LIN {X 0,Y 573.173,Z 473.905,A -85,B 0,C 180,E1 -2067.979,E2 -2067.979} C_VEL
LIN {X 0,Y 573.326,Z 473.883,A -85,B 0,C 180,E1 -2070,E2 -2070} C_VEL
LIN {X 0,Y 573.306,Z 473.888,A -85,B 0,C 180,E1 -2072.81,E2 -2072.81} C_VEL
LIN {X 0,Y 573.299,Z 473.886,A -85,B 0,C 180,E1 -2075.628,E2 -2075.628} C_VEL
LIN {X 0,Y 573.287,Z 473.888,A -85,B 0,C 180,E1 -2078.459,E2 -2078.459} C_VEL
LIN {X 0,Y 573.274,Z 473.891,A -85,B 0,C 180,E1 -2081.312,E2 -2081.312} C_VEL
LIN {X 0,Y 573.283,Z 473.889,A -85,B 0,C 180,E1 -2084.424,E2 -2084.424} C_VEL
LIN {X 0,Y 573.261,Z 473.893,A -85,B 0,C 180,E1 -2087.111,E2 -2087.111} C_VEL
LIN {X 0,Y 573.255,Z 473.892,A -85,B 0,C 180,E1 -2090.076,E2 -2090.076} C_VEL
LIN {X 0,Y 573.235,Z 473.896,A -85,B 0,C 180,E1 -2093.099,E2 -2093.099} C_VEL
LIN {X 0,Y 573.258,Z 473.894,A -85,B 0,C 180,E1 -2095.409,E2 -2095.409} C_VEL
LIN {X 0,Y 573.253,Z 473.893,A -85,B 0,C 180,E1 -2098.029,E2 -2098.029} C_VEL
LIN {X 0,Y 573.246,Z 473.893,A -85,B 0,C 180,E1 -2100.885,E2 -2100.885} C_VEL
LIN {X 0,Y 573.262,Z 473.893,A -85,B 0,C 180,E1 -2103.524,E2 -2103.524} C_VEL
LIN {X 0,Y 573.261,Z 473.894,A -85,B 0,C 180,E1 -2106.048,E2 -2106.048} C_VEL
LIN {X 0,Y 573.249,Z 473.892,A -85,B 0,C 180,E1 -2108.7,E2 -2108.7} C_VEL
LIN {X 0,Y 573.228,Z 473.895,A -85,B 0,C 180,E1 -2111.457,E2 -2111.457} C_VEL
LIN {X 0,Y 573.238,Z 473.896,A -85,B 0,C 180,E1 -2114.333,E2 -2114.333} C_VEL
LIN {X 0,Y 573.243,Z 473.893,A -85,B 0,C 180,E1 -2117.358,E2 -2117.358} C_VEL
LIN {X 0,Y 573.273,Z 473.889,A -85,B 0,C 180,E1 -2119.477,E2 -2119.477} C_VEL
LIN {X 0,Y 573.235,Z 473.895,A -85,B 0,C 180,E1 -2122.192,E2 -2122.192} C_VEL
LIN {X 0,Y 573.236,Z 473.894,A -85,B 0,C 180,E1 -2125.228,E2 -2125.228} C_VEL
LIN {X 0,Y 573.256,Z 473.891,A -85,B 0,C 180,E1 -2127.77,E2 -2127.77} C_VEL
LIN {X 0,Y 573.263,Z 473.893,A -85,B 0,C 180,E1 -2130.634,E2 -2130.634} C_VEL
LIN {X 0,Y 573.27,Z 473.89,A -85,B 0,C 180,E1 -2133.5,E2 -2133.5} C_VEL
LIN {X 0,Y 573.23,Z 473.895,A -85,B 0,C 180,E1 -2136.134,E2 -2136.134} C_VEL
LIN {X 0,Y 573.26,Z 473.893,A -85,B 0,C 180,E1 -2139.174,E2 -2139.174} C_VEL
LIN {X 0,Y 573.229,Z 473.898,A -85,B 0,C 180,E1 -2141.411,E2 -2141.411} C_VEL
LIN {X 0,Y 573.253,Z 473.893,A -85,B 0,C 180,E1 -2143.622,E2 -2143.622} C_VEL
LIN {X 0,Y 573.272,Z 473.89,A -85,B 0,C 180,E1 -2145.807,E2 -2145.807} C_VEL
LIN {X 0,Y 573.261,Z 473.892,A -85,B 0,C 180,E1 -2148.745,E2 -2148.745} C_VEL
LIN {X 0,Y 573.29,Z 473.887,A -85,B 0,C 180,E1 -2151.541,E2 -2151.541} C_VEL
LIN {X 0,Y 573.289,Z 473.891,A -85,B 0,C 180,E1 -2154.372,E2 -2154.372} C_VEL
LIN {X 0,Y 573.312,Z 473.887,A -85,B 0,C 180,E1 -2157.892,E2 -2157.892} C_VEL
LIN {X 0,Y 573.332,Z 473.882,A -85,B 0,C 180,E1 -2160.702,E2 -2160.702} C_VEL
LIN {X 0,Y 573.24,Z 473.894,A -85,B 0,C 180,E1 -2163.514,E2 -2163.514} C_VEL
LIN {X 0,Y 573.294,Z 473.887,A -85,B 0,C 180,E1 -2165.628,E2 -2165.628} C_VEL
LIN {X 0,Y 573.288,Z 473.89,A -85,B 0,C 180,E1 -2168.459,E2 -2168.459} C_VEL
LIN {X 0,Y 573.27,Z 473.89,A -85,B 0,C 180,E1 -2171.312,E2 -2171.312} C_VEL
LIN {X 0,Y 573.271,Z 473.89,A -85,B 0,C 180,E1 -2174.193,E2 -2174.193} C_VEL
LIN {X 0,Y 573.259,Z 473.892,A -85,B 0,C 180,E1 -2177.112,E2 -2177.112} C_VEL
LIN {X 0,Y 573.251,Z 473.893,A -85,B 0,C 180,E1 -2180.077,E2 -2180.077} C_VEL
LIN {X 0,Y 573.232,Z 473.895,A -85,B 0,C 180,E1 -2183.099,E2 -2183.099} C_VEL
LIN {X 0,Y 573.253,Z 473.893,A -85,B 0,C 180,E1 -2185.41,E2 -2185.41} C_VEL
LIN {X 0,Y 573.251,Z 473.892,A -85,B 0,C 180,E1 -2188.03,E2 -2188.03} C_VEL
LIN {X 0,Y 573.255,Z 473.892,A -85,B 0,C 180,E1 -2190.176,E2 -2190.176} C_VEL
LIN {X 0,Y 573.255,Z 473.891,A -85,B 0,C 180,E1 -2192.645,E2 -2192.645} C_VEL
LIN {X 0,Y 573.267,Z 473.89,A -85,B 0,C 180,E1 -2195.184,E2 -2195.184} C_VEL
LIN {X 0,Y 573.236,Z 473.895,A -85,B 0,C 180,E1 -2197.807,E2 -2197.807} C_VEL
LIN {X 0,Y 573.268,Z 473.893,A -85,B 0,C 180,E1 -2200.528,E2 -2200.528} C_VEL
LIN {X 0,Y 573.254,Z 473.892,A -85,B 0,C 180,E1 -2203.671,E2 -2203.671} C_VEL
LIN {X 0,Y 573.238,Z 473.895,A -85,B 0,C 180,E1 -2206.641,E2 -2206.641} C_VEL
LIN {X 0,Y 573.272,Z 473.89,A -85,B 0,C 180,E1 -2209.478,E2 -2209.478} C_VEL
LIN {X 0,Y 573.235,Z 473.896,A -85,B 0,C 180,E1 -2212.193,E2 -2212.193} C_VEL
LIN {X 0,Y 573.269,Z 473.892,A -85,B 0,C 180,E1 -2214.817,E2 -2214.817} C_VEL
LIN {X 0,Y 573.253,Z 473.894,A -85,B 0,C 180,E1 -2217.355,E2 -2217.355} C_VEL
LIN {X 0,Y 573.27,Z 473.92,A -85,B 0,C 180,E1 -2218.113,E2 -2218.113} C_VEL
LIN {X 0,Y 573.657,Z 478.198,A -85,B 0,C 180,E1 -2219.447,E2 -2219.447} C_VEL
LIN {X 0,Y 573.521,Z 487.647,A -85,B 0,C 180,E1 -2222.248,E2 -2222.248} C_VEL
LIN {X 0,Y 573.466,Z 497.583,A -85,B 0,C 180,E1 -2225.079,E2 -2225.079} C_VEL
LIN {X 0,Y 573.37,Z 508.135,A -85,B 0,C 180,E1 -2228.047,E2 -2228.047} C_VEL
LIN {X 0,Y 573.251,Z 519.115,A -85,B 0,C 180,E1 -2231.072,E2 -2231.072} C_VEL
LIN {X 0,Y 573.175,Z 529.877,A -85,B 0,C 180,E1 -2233.986,E2 -2233.986} C_VEL
LIN {X 0,Y 573.105,Z 540.748,A -85,B 0,C 180,E1 -2236.888,E2 -2236.888} C_VEL
LIN {X 0,Y 573.057,Z 550.26,A -85,B 0,C 180,E1 -2239.4,E2 -2239.4} C_VEL
LIN {X 0,Y 573.08,Z 553.109,A -85,B 0,C 180,E1 -2240.125,E2 -2240.125} C_VEL
LIN {X 0,Y 573.479,Z 559.596,A -85,B 0,C 180,E1 -2240.277,E2 -2240.277} C_VEL
LIN {X 0,Y 573.449,Z 568.903,A -85,B 0,C 180,E1 -2240.566,E2 -2240.566} C_VEL
LIN {X 0,Y 573.402,Z 577.409,A -85,B 0,C 180,E1 -2240.921,E2 -2240.921} C_VEL
LIN {X 0,Y 573.339,Z 585.736,A -85,B 0,C 180,E1 -2241.364,E2 -2241.364} C_VEL
LIN {X 0,Y 573.252,Z 593.772,A -85,B 0,C 180,E1 -2241.895,E2 -2241.895} C_VEL
LIN {X 0,Y 573.187,Z 601.421,A -85,B 0,C 180,E1 -2242.515,E2 -2242.515} C_VEL
LIN {X 0,Y 573.155,Z 609.552,A -85,B 0,C 180,E1 -2243.323,E2 -2243.323} C_VEL
LIN {X 0,Y 573.112,Z 616.435,A -85,B 0,C 180,E1 -2244.194,E2 -2244.194} C_VEL
LIN {X 0,Y 573.005,Z 621.989,A -85,B 0,C 180,E1 -2245.075,E2 -2245.075} C_VEL
LIN {X 0,Y 573.036,Z 627.149,A -85,B 0,C 180,E1 -2246.133,E2 -2246.133} C_VEL
LIN {X 0,Y 572.992,Z 629.79,A -85,B 0,C 180,E1 -2246.836,E2 -2246.836} C_VEL
LIN {X 0,Y 572.939,Z 632.682,A -85,B 0,C 180,E1 -2247.891,E2 -2247.891} C_VEL
LIN {X 0,Y 572.945,Z 633.937,A -85,B 0,C 180,E1 -2248.595,E2 -2248.595} C_VEL
LIN {X 0,Y 572.938,Z 634.711,A -85,B 0,C 180,E1 -2249.298,E2 -2249.298} C_VEL
LIN {X 0,Y 572.935,Z 635,A -85,B 0,C 180,E1 -2250,E2 -2250} C_VEL
LIN {X 0,Y 572.938,Z 634.711,A -85,B 0,C 180,E1 -2250.703,E2 -2250.703} C_VEL
LIN {X 0,Y 572.945,Z 633.936,A -85,B 0,C 180,E1 -2251.406,E2 -2251.406} C_VEL
LIN {X 0,Y 572.939,Z 632.68,A -85,B 0,C 180,E1 -2252.109,E2 -2252.109} C_VEL
LIN {X 0,Y 572.992,Z 629.787,A -85,B 0,C 180,E1 -2253.164,E2 -2253.164} C_VEL
LIN {X 0,Y 573.024,Z 627.146,A -85,B 0,C 180,E1 -2253.868,E2 -2253.868} C_VEL
LIN {X 0,Y 573.005,Z 621.984,A -85,B 0,C 180,E1 -2254.926,E2 -2254.926} C_VEL
LIN {X 0,Y 573.137,Z 615.184,A -85,B 0,C 180,E1 -2255.983,E2 -2255.983} C_VEL
LIN {X 0,Y 573.164,Z 607.801,A -85,B 0,C 180,E1 -2256.86,E2 -2256.86} C_VEL
LIN {X 0,Y 573.213,Z 600.402,A -85,B 0,C 180,E1 -2257.574,E2 -2257.574} C_VEL
LIN {X 0,Y 573.275,Z 592.542,A -85,B 0,C 180,E1 -2258.194,E2 -2258.194} C_VEL
LIN {X 0,Y 573.385,Z 582.727,A -85,B 0,C 180,E1 -2258.814,E2 -2258.814} C_VEL
LIN {X 0,Y 573.429,Z 571.291,A -85,B 0,C 180,E1 -2259.346,E2 -2259.346} C_VEL
LIN {X 0,Y 573.507,Z 561.233,A -85,B 0,C 180,E1 -2259.679,E2 -2259.679} C_VEL
LIN {X 0,Y 573.212,Z 555.017,A -85,B 0,C 180,E1 -2259.84,E2 -2259.84} C_VEL
LIN {X 0,Y 573.019,Z 553.301,A -85,B 0,C 180,E1 -2259.887,E2 -2259.887} C_VEL
LIN {X 0,Y 573.067,Z 544.36,A -85,B 0,C 180,E1 -2262.393,E2 -2262.393} C_VEL
LIN {X 0,Y 573.155,Z 534.141,A -85,B 0,C 180,E1 -2265.286,E2 -2265.286} C_VEL
LIN {X 0,Y 573.21,Z 523.922,A -85,B 0,C 180,E1 -2268.219,E2 -2268.219} C_VEL
LIN {X 0,Y 573.273,Z 514.981,A -85,B 0,C 180,E1 -2270.826,E2 -2270.826} C_VEL
LIN {X 0,Y 573.346,Z 506.041,A -85,B 0,C 180,E1 -2273.477,E2 -2273.477} C_VEL
LIN {X 0,Y 573.412,Z 496.934,A -85,B 0,C 180,E1 -2276.183,E2 -2276.183} C_VEL
LIN {X 0,Y 573.474,Z 487.899,A -85,B 0,C 180,E1 -2278.952,E2 -2278.952} C_VEL
LIN {X 0,Y 573.623,Z 480.281,A -85,B 0,C 180,E1 -2281.38,E2 -2281.38} C_VEL
LIN {X 0,Y 573.54,Z 475.462,A -85,B 0,C 180,E1 -2283.045,E2 -2283.045} C_VEL
LIN {X 0,Y 573.29,Z 473.89,A -85,B 0,C 180,E1 -2283.692,E2 -2283.692} C_VEL
LIN {X 0,Y 573.24,Z 473.893,A -85,B 0,C 180,E1 -2286.05,E2 -2286.05} C_VEL
LIN {X 0,Y 573.25,Z 473.896,A -85,B 0,C 180,E1 -2288.701,E2 -2288.701} C_VEL
LIN {X 0,Y 573.232,Z 473.894,A -85,B 0,C 180,E1 -2291.457,E2 -2291.457} C_VEL
LIN {X 0,Y 573.238,Z 473.891,A -85,B 0,C 180,E1 -2294.334,E2 -2294.334} C_VEL
LIN {X 0,Y 573.246,Z 473.89,A -85,B 0,C 180,E1 -2297.358,E2 -2297.358} C_VEL
LIN {X 0,Y 573.243,Z 473.891,A -85,B 0,C 180,E1 -2300.393,E2 -2300.393} C_VEL
LIN {X 0,Y 573.255,Z 473.894,A -85,B 0,C 180,E1 -2303.078,E2 -2303.078} C_VEL
LIN {X 0,Y 573.269,Z 473.889,A -85,B 0,C 180,E1 -2305.672,E2 -2305.672} C_VEL
LIN {X 0,Y 573.141,Z 473.909,A -85,B 0,C 180,E1 -2308.178,E2 -2308.178} C_VEL
LIN {X 0,Y 573.099,Z 477.229,A -85,B 0,C 180,E1 -2310.625,E2 -2310.625} C_VEL
LIN {X 0,Y 573.045,Z 480.484,A -85,B 0,C 180,E1 -2313.014,E2 -2313.014} C_VEL
LIN {X 0,Y 573.025,Z 483.626,A -85,B 0,C 180,E1 -2315.355,E2 -2315.355} C_VEL
LIN {X 0,Y 572.985,Z 486.997,A -85,B 0,C 180,E1 -2317.652,E2 -2317.652} C_VEL
LIN {X 0,Y 573.021,Z 491.592,A -85,B 0,C 180,E1 -2320.661,E2 -2320.661} C_VEL
LIN {X 0,Y 572.976,Z 496.187,A -85,B 0,C 180,E1 -2323.614,E2 -2323.614} C_VEL
LIN {X 0,Y 572.993,Z 500.783,A -85,B 0,C 180,E1 -2326.524,E2 -2326.524} C_VEL
LIN {X 0,Y 572.98,Z 505.378,A -85,B 0,C 180,E1 -2329.398,E2 -2329.398} C_VEL
LIN {X 0,Y 572.976,Z 506.707,A -85,B 0,C 180,E1 -2330.224,E2 -2330.224} C_VEL
LIN {X 0,Y 573.49,Z 512.89,A -85,B 0,C 180,E1 -2330.411,E2 -2330.411} C_VEL
LIN {X 0,Y 573.429,Z 524.583,A -85,B 0,C 180,E1 -2330.832,E2 -2330.832} C_VEL
LIN {X 0,Y 573.333,Z 534.974,A -85,B 0,C 180,E1 -2331.364,E2 -2331.364} C_VEL
LIN {X 0,Y 573.246,Z 543.153,A -85,B 0,C 180,E1 -2331.895,E2 -2331.895} C_VEL
LIN {X 0,Y 573.196,Z 550.906,A -85,B 0,C 180,E1 -2332.515,E2 -2332.515} C_VEL
LIN {X 0,Y 573.167,Z 557.376,A -85,B 0,C 180,E1 -2333.141,E2 -2333.141} C_VEL
LIN {X 0,Y 573.138,Z 564.834,A -85,B 0,C 180,E1 -2334.017,E2 -2334.017} C_VEL
LIN {X 0,Y 573.004,Z 571.741,A -85,B 0,C 180,E1 -2335.075,E2 -2335.075} C_VEL
LIN {X 0,Y 573.033,Z 575.438,A -85,B 0,C 180,E1 -2335.78,E2 -2335.78} C_VEL
LIN {X 0,Y 573.053,Z 578.452,A -85,B 0,C 180,E1 -2336.484,E2 -2336.484} C_VEL
LIN {X 0,Y 572.962,Z 580.787,A -85,B 0,C 180,E1 -2337.188,E2 -2337.188} C_VEL
LIN {X 0,Y 572.937,Z 582.578,A -85,B 0,C 180,E1 -2337.891,E2 -2337.891} C_VEL
LIN {X 0,Y 572.946,Z 583.874,A -85,B 0,C 180,E1 -2338.594,E2 -2338.594} C_VEL
LIN {X 0,Y 572.937,Z 584.69,A -85,B 0,C 180,E1 -2339.297,E2 -2339.297} C_VEL
LIN {X 0,Y 572.934,Z 584.996,A -85,B 0,C 180,E1 -2340,E2 -2340} C_VEL
LIN {X 0,Y 572.939,Z 584.731,A -85,B 0,C 180,E1 -2340.703,E2 -2340.703} C_VEL
LIN {X 0,Y 572.945,Z 583.997,A -85,B 0,C 180,E1 -2341.406,E2 -2341.406} C_VEL
LIN {X 0,Y 572.939,Z 582.783,A -85,B 0,C 180,E1 -2342.109,E2 -2342.109} C_VEL
LIN {X 0,Y 572.98,Z 579.935,A -85,B 0,C 180,E1 -2343.164,E2 -2343.164} C_VEL
LIN {X 0,Y 573.026,Z 577.341,A -85,B 0,C 180,E1 -2343.868,E2 -2343.868} C_VEL
LIN {X 0,Y 572.984,Z 572.231,A -85,B 0,C 180,E1 -2344.925,E2 -2344.925} C_VEL
LIN {X 0,Y 573.113,Z 566.733,A -85,B 0,C 180,E1 -2345.807,E2 -2345.807} C_VEL
LIN {X 0,Y 573.157,Z 558.342,A -85,B 0,C 180,E1 -2346.849,E2 -2346.849} C_VEL
LIN {X 0,Y 573.213,Z 550.917,A -85,B 0,C 180,E1 -2347.574,E2 -2347.574} C_VEL
LIN {X 0,Y 573.274,Z 543.167,A -85,B 0,C 180,E1 -2348.194,E2 -2348.194} C_VEL
LIN {X 0,Y 573.386,Z 534.991,A -85,B 0,C 180,E1 -2348.724,E2 -2348.724} C_VEL
LIN {X 0,Y 573.394,Z 526.474,A -85,B 0,C 180,E1 -2349.169,E2 -2349.169} C_VEL
LIN {X 0,Y 573.488,Z 515.241,A -85,B 0,C 180,E1 -2349.612,E2 -2349.612} C_VEL
LIN {X 0,Y 573.182,Z 508.35,A -85,B 0,C 180,E1 -2349.806,E2 -2349.806} C_VEL
LIN {X 0,Y 572.968,Z 506.482,A -85,B 0,C 180,E1 -2349.888,E2 -2349.888} C_VEL
LIN {X 0,Y 572.967,Z 501.591,A -85,B 0,C 180,E1 -2352.755,E2 -2352.755} C_VEL
LIN {X 0,Y 572.988,Z 497.923,A -85,B 0,C 180,E1 -2354.926,E2 -2354.926} C_VEL
LIN {X 0,Y 572.967,Z 493.032,A -85,B 0,C 180,E1 -2357.857,E2 -2357.857} C_VEL
LIN {X 0,Y 572.998,Z 489.364,A -85,B 0,C 180,E1 -2360.086,E2 -2360.086} C_VEL
LIN {X 0,Y 573,Z 488.115,A -85,B 0,C 180,E1 -2360.852,E2 -2360.852} C_VEL
LIN {X 0,Y 572.335,Z 487.218,A -85,B 0,C 180,E1 -2361.432,E2 -2361.432} C_VEL
LIN {X 0,Y 569.468,Z 485.896,A -85,B 0,C 180,E1 -2362.375,E2 -2362.375} C_VEL
LIN {X 0,Y 567.048,Z 484.865,A -85,B 0,C 180,E1 -2363.135,E2 -2363.135} C_VEL
LIN {X 0,Y 566.015,Z 484.027,A -85,B 0,C 180,E1 -2363.72,E2 -2363.72} C_VEL
LIN {X 0,Y 565.934,Z 483.727,A -85,B 0,C 180,E1 -2363.918,E2 -2363.918} C_VEL
LIN {X 0,Y 566.026,Z 479.241,A -85,B 0,C 180,E1 -2366.912,E2 -2366.912} C_VEL
LIN {X 0,Y 566.051,Z 478.708,A -85,B 0,C 180,E1 -2367.293,E2 -2367.293} C_VEL
LIN {X 0,Y 566.076,Z 484.914,A -85,B 0,C 180,E1 -2369.776,E2 -2369.776} C_VEL
LIN {X 0,Y 566.114,Z 491.47,A -85,B 0,C 180,E1 -2372.415,E2 -2372.415} C_VEL
LIN {X 0,Y 566.048,Z 497.672,A -85,B 0,C 180,E1 -2374.97,E2 -2374.97} C_VEL
LIN {X 0,Y 566.002,Z 504.801,A -85,B 0,C 180,E1 -2377.926,E2 -2377.926} C_VEL
LIN {X 0,Y 565.959,Z 511.741,A -85,B 0,C 180,E1 -2380.756,E2 -2380.756} C_VEL
LIN {X 0,Y 565.94,Z 518.557,A -85,B 0,C 180,E1 -2383.5,E2 -2383.5} C_VEL
LIN {X 0,Y 565.921,Z 525.026,A -85,B 0,C 180,E1 -2386.078,E2 -2386.078} C_VEL
LIN {X 0,Y 566.504,Z 532.234,A -85,B 0,C 180,E1 -2386.273,E2 -2386.273} C_VEL
LIN {X 0,Y 566.445,Z 541.756,A -85,B 0,C 180,E1 -2386.602,E2 -2386.602} C_VEL
LIN {X 0,Y 566.326,Z 552.862,A -85,B 0,C 180,E1 -2387.126,E2 -2387.126} C_VEL
LIN {X 0,Y 566.235,Z 563.213,A -85,B 0,C 180,E1 -2387.794,E2 -2387.794} C_VEL
LIN {X 0,Y 566.159,Z 571.873,A -85,B 0,C 180,E1 -2388.504,E2 -2388.504} C_VEL
LIN {X 0,Y 566.031,Z 580.29,A -85,B 0,C 180,E1 -2389.375,E2 -2389.375} C_VEL
LIN {X 0,Y 565.996,Z 587.634,A -85,B 0,C 180,E1 -2390.341,E2 -2390.341} C_VEL
LIN {X 0,Y 565.922,Z 594.266,A -85,B 0,C 180,E1 -2391.479,E2 -2391.479} C_VEL
LIN {X 0,Y 565.906,Z 599.119,A -85,B 0,C 180,E1 -2392.638,E2 -2392.638} C_VEL
LIN {X 0,Y 565.859,Z 602.529,A -85,B 0,C 180,E1 -2393.833,E2 -2393.833} C_VEL
LIN {X 0,Y 565.849,Z 604.519,A -85,B 0,C 180,E1 -2395.059,E2 -2395.059} C_VEL
LIN {X 0,Y 565.85,Z 604.904,A -85,B 0,C 180,E1 -2396.321,E2 -2396.321} C_VEL
LIN {X 0,Y 565.826,Z 604.648,A -85,B 0,C 180,E1 -2396.871,E2 -2396.871} C_VEL
LIN {X 0,Y 565.853,Z 603.582,A -85,B 0,C 180,E1 -2397.719,E2 -2397.719} C_VEL
LIN {X 0,Y 565.898,Z 600.701,A -85,B 0,C 180,E1 -2398.973,E2 -2398.973} C_VEL
LIN {X 0,Y 565.908,Z 597.854,A -85,B 0,C 180,E1 -2399.803,E2 -2399.803} C_VEL
LIN {X 0,Y 565.95,Z 593.777,A -85,B 0,C 180,E1 -2400.705,E2 -2400.705} C_VEL
LIN {X 0,Y 565.974,Z 588.203,A -85,B 0,C 180,E1 -2401.663,E2 -2401.663} C_VEL
LIN {X 0,Y 566.056,Z 582.479,A -85,B 0,C 180,E1 -2402.452,E2 -2402.452} C_VEL
LIN {X 0,Y 566.094,Z 574.222,A -85,B 0,C 180,E1 -2403.364,E2 -2403.364} C_VEL
LIN {X 0,Y 566.169,Z 566.419,A -85,B 0,C 180,E1 -2404.051,E2 -2404.051} C_VEL
LIN {X 0,Y 566.267,Z 558.201,A -85,B 0,C 180,E1 -2404.638,E2 -2404.638} C_VEL
LIN {X 0,Y 566.343,Z 549.386,A -85,B 0,C 180,E1 -2405.142,E2 -2405.142} C_VEL
LIN {X 0,Y 566.465,Z 540.46,A -85,B 0,C 180,E1 -2405.539,E2 -2405.539} C_VEL
LIN {X 0,Y 566.5,Z 530.802,A -85,B 0,C 180,E1 -2405.857,E2 -2405.857} C_VEL
LIN {X 0,Y 565.895,Z 525.251,A -85,B 0,C 180,E1 -2406.024,E2 -2406.024} C_VEL
LIN {X 0,Y 565.906,Z 518.495,A -85,B 0,C 180,E1 -2408.89,E2 -2408.89} C_VEL
LIN {X 0,Y 565.962,Z 513.187,A -85,B 0,C 180,E1 -2411.164,E2 -2411.164} C_VEL
LIN {X 0,Y 565.98,Z 506.312,A -85,B 0,C 180,E1 -2414.146,E2 -2414.146} C_VEL
LIN {X 0,Y 566.01,Z 501.294,A -85,B 0,C 180,E1 -2416.354,E2 -2416.354} C_VEL
LIN {X 0,Y 566.056,Z 494.758,A -85,B 0,C 180,E1 -2419.266,E2 -2419.266} C_VEL
LIN {X 0,Y 566.065,Z 488.079,A -85,B 0,C 180,E1 -2422.15,E2 -2422.15} C_VEL
LIN {X 0,Y 566.126,Z 481.423,A -85,B 0,C 180,E1 -2425.014,E2 -2425.014} C_VEL
LIN {X 0,Y 566.113,Z 474.784,A -85,B 0,C 180,E1 -2427.954,E2 -2427.954} C_VEL
LIN {X 0,Y 566.296,Z 474.758,A -85,B 0,C 180,E1 -2430,E2 -2430} C_VEL
LIN {X 0,Y 566.272,Z 474.764,A -85,B 0,C 180,E1 -2432.845,E2 -2432.845} C_VEL
LIN {X 0,Y 566.267,Z 474.762,A -85,B 0,C 180,E1 -2435.698,E2 -2435.698} C_VEL
LIN {X 0,Y 566.23,Z 474.768,A -85,B 0,C 180,E1 -2438.565,E2 -2438.565} C_VEL
LIN {X 0,Y 566.244,Z 474.766,A -85,B 0,C 180,E1 -2441.454,E2 -2441.454} C_VEL
LIN {X 0,Y 566.236,Z 474.767,A -85,B 0,C 180,E1 -2444.506,E2 -2444.506} C_VEL
LIN {X 0,Y 566.205,Z 474.771,A -85,B 0,C 180,E1 -2447.331,E2 -2447.331} C_VEL
LIN {X 0,Y 566.216,Z 474.769,A -85,B 0,C 180,E1 -2450.337,E2 -2450.337} C_VEL
LIN {X 0,Y 566.191,Z 474.771,A -85,B 0,C 180,E1 -2453.403,E2 -2453.403} C_VEL
LIN {X 0,Y 566.226,Z 474.767,A -85,B 0,C 180,E1 -2455.748,E2 -2455.748} C_VEL
LIN {X 0,Y 566.202,Z 474.77,A -85,B 0,C 180,E1 -2458.202,E2 -2458.202} C_VEL
LIN {X 0,Y 566.196,Z 474.771,A -85,B 0,C 180,E1 -2460.591,E2 -2460.591} C_VEL
LIN {X 0,Y 566.23,Z 474.766,A -85,B 0,C 180,E1 -2463.101,E2 -2463.101} C_VEL
LIN {X 0,Y 566.213,Z 474.769,A -85,B 0,C 180,E1 -2465.688,E2 -2465.688} C_VEL
LIN {X 0,Y 566.217,Z 474.769,A -85,B 0,C 180,E1 -2468.559,E2 -2468.559} C_VEL
LIN {X 0,Y 566.202,Z 474.77,A -85,B 0,C 180,E1 -2471.137,E2 -2471.137} C_VEL
LIN {X 0,Y 566.199,Z 474.772,A -85,B 0,C 180,E1 -2474.035,E2 -2474.035} C_VEL
LIN {X 0,Y 566.204,Z 474.769,A -85,B 0,C 180,E1 -2477.082,E2 -2477.082} C_VEL
LIN {X 0,Y 566.226,Z 474.767,A -85,B 0,C 180,E1 -2479.802,E2 -2479.802} C_VEL
LIN {X 0,Y 566.197,Z 474.773,A -85,B 0,C 180,E1 -2482.599,E2 -2482.599} C_VEL
LIN {X 0,Y 566.198,Z 474.771,A -85,B 0,C 180,E1 -2485.181,E2 -2485.181} C_VEL
LIN {X 0,Y 566.235,Z 474.766,A -85,B 0,C 180,E1 -2487.744,E2 -2487.744} C_VEL
LIN {X 0,Y 566.202,Z 474.77,A -85,B 0,C 180,E1 -2490.328,E2 -2490.328} C_VEL
LIN {X 0,Y 566.224,Z 474.767,A -85,B 0,C 180,E1 -2492.661,E2 -2492.661} C_VEL
LIN {X 0,Y 566.234,Z 474.765,A -85,B 0,C 180,E1 -2495.039,E2 -2495.039} C_VEL
LIN {X 0,Y 566.195,Z 474.772,A -85,B 0,C 180,E1 -2498.137,E2 -2498.137} C_VEL
LIN {X 0,Y 566.236,Z 474.766,A -85,B 0,C 180,E1 -2500.611,E2 -2500.611} C_VEL
LIN {X 0,Y 566.216,Z 474.768,A -85,B 0,C 180,E1 -2503.412,E2 -2503.412} C_VEL
LIN {X 0,Y 566.199,Z 474.771,A -85,B 0,C 180,E1 -2506.359,E2 -2506.359} C_VEL
LIN {X 0,Y 566.232,Z 474.768,A -85,B 0,C 180,E1 -2508.675,E2 -2508.675} C_VEL
LIN {X 0,Y 566.233,Z 474.766,A -85,B 0,C 180,E1 -2511.434,E2 -2511.434} C_VEL
LIN {X 0,Y 566.257,Z 474.766,A -85,B 0,C 180,E1 -2514.302,E2 -2514.302} C_VEL
LIN {X 0,Y 566.282,Z 474.763,A -85,B 0,C 180,E1 -2517.866,E2 -2517.866} C_VEL
LIN {X 0,Y 566.303,Z 474.757,A -85,B 0,C 180,E1 -2520.711,E2 -2520.711} C_VEL
LIN {X 0,Y 566.276,Z 474.763,A -85,B 0,C 180,E1 -2522.845,E2 -2522.845} C_VEL
LIN {X 0,Y 566.262,Z 474.763,A -85,B 0,C 180,E1 -2525.698,E2 -2525.698} C_VEL
LIN {X 0,Y 566.232,Z 474.769,A -85,B 0,C 180,E1 -2528.566,E2 -2528.566} C_VEL
LIN {X 0,Y 566.24,Z 474.765,A -85,B 0,C 180,E1 -2531.454,E2 -2531.454} C_VEL
LIN {X 0,Y 566.232,Z 474.769,A -85,B 0,C 180,E1 -2534.507,E2 -2534.507} C_VEL
LIN {X 0,Y 566.203,Z 474.77,A -85,B 0,C 180,E1 -2537.331,E2 -2537.331} C_VEL
LIN {X 0,Y 566.212,Z 474.772,A -85,B 0,C 180,E1 -2540.337,E2 -2540.337} C_VEL
LIN {X 0,Y 566.189,Z 474.772,A -85,B 0,C 180,E1 -2543.404,E2 -2543.404} C_VEL
LIN {X 0,Y 566.212,Z 474.769,A -85,B 0,C 180,E1 -2545.749,E2 -2545.749} C_VEL
LIN {X 0,Y 566.2,Z 474.77,A -85,B 0,C 180,E1 -2548.202,E2 -2548.202} C_VEL
LIN {X 0,Y 566.192,Z 474.771,A -85,B 0,C 180,E1 -2550.592,E2 -2550.592} C_VEL
LIN {X 0,Y 566.227,Z 474.767,A -85,B 0,C 180,E1 -2553.102,E2 -2553.102} C_VEL
LIN {X 0,Y 566.211,Z 474.772,A -85,B 0,C 180,E1 -2555.689,E2 -2555.689} C_VEL
LIN {X 0,Y 566.21,Z 474.769,A -85,B 0,C 180,E1 -2558.559,E2 -2558.559} C_VEL
LIN {X 0,Y 566.21,Z 474.769,A -85,B 0,C 180,E1 -2561.136,E2 -2561.136} C_VEL
LIN {X 0,Y 566.2,Z 474.773,A -85,B 0,C 180,E1 -2564.035,E2 -2564.035} C_VEL
LIN {X 0,Y 566.2,Z 474.77,A -85,B 0,C 180,E1 -2567.083,E2 -2567.083} C_VEL
LIN {X 0,Y 566.226,Z 474.769,A -85,B 0,C 180,E1 -2569.803,E2 -2569.803} C_VEL
LIN {X 0,Y 566.198,Z 474.772,A -85,B 0,C 180,E1 -2572.599,E2 -2572.599} C_VEL
LIN {X 0,Y 566.221,Z 474.768,A -85,B 0,C 180,E1 -2575.184,E2 -2575.184} C_VEL
LIN {X 0,Y 566.249,Z 474.83,A -85,B 0,C 180,E1 -2577.955,E2 -2577.955} C_VEL
LIN {X 0,Y 566.698,Z 479.52,A -85,B 0,C 180,E1 -2579.439,E2 -2579.439} C_VEL
LIN {X 0,Y 566.549,Z 490.329,A -85,B 0,C 180,E1 -2582.679,E2 -2582.679} C_VEL
LIN {X 0,Y 566.404,Z 501.314,A -85,B 0,C 180,E1 -2585.829,E2 -2585.829} C_VEL
LIN {X 0,Y 566.288,Z 510.978,A -85,B 0,C 180,E1 -2588.56,E2 -2588.56} C_VEL
LIN {X 0,Y 566.21,Z 520.365,A -85,B 0,C 180,E1 -2591.173,E2 -2591.173} C_VEL
LIN {X 0,Y 566.111,Z 529.877,A -85,B 0,C 180,E1 -2593.78,E2 -2593.78} C_VEL
LIN {X 0,Y 566.04,Z 539.389,A -85,B 0,C 180,E1 -2596.355,E2 -2596.355} C_VEL
LIN {X 0,Y 566.046,Z 548.403,A -85,B 0,C 180,E1 -2598.772,E2 -2598.772} C_VEL
LIN {X 0,Y 565.98,Z 552.978,A -85,B 0,C 180,E1 -2599.989,E2 -2599.989} C_VEL
LIN {X 0,Y 566.495,Z 559.596,A -85,B 0,C 180,E1 -2600.156,E2 -2600.156} C_VEL
LIN {X 0,Y 566.459,Z 568.901,A -85,B 0,C 180,E1 -2600.448,E2 -2600.448} C_VEL
LIN {X 0,Y 566.4,Z 577.407,A -85,B 0,C 180,E1 -2600.808,E2 -2600.808} C_VEL
LIN {X 0,Y 566.32,Z 585.737,A -85,B 0,C 180,E1 -2601.256,E2 -2601.256} C_VEL
LIN {X 0,Y 566.209,Z 593.774,A -85,B 0,C 180,E1 -2601.794,E2 -2601.794} C_VEL
LIN {X 0,Y 566.124,Z 602.435,A -85,B 0,C 180,E1 -2602.511,E2 -2602.511} C_VEL
LIN {X 0,Y 566.064,Z 610.384,A -85,B 0,C 180,E1 -2603.336,E2 -2603.336} C_VEL
LIN {X 0,Y 566.057,Z 616.436,A -85,B 0,C 180,E1 -2604.121,E2 -2604.121} C_VEL
LIN {X 0,Y 565.913,Z 621.99,A -85,B 0,C 180,E1 -2605.013,E2 -2605.013} C_VEL
LIN {X 0,Y 565.944,Z 627.15,A -85,B 0,C 180,E1 -2606.084,E2 -2606.084} C_VEL
LIN {X 0,Y 565.914,Z 629.79,A -85,B 0,C 180,E1 -2606.797,E2 -2606.797} C_VEL
LIN {X 0,Y 565.84,Z 632.682,A -85,B 0,C 180,E1 -2607.865,E2 -2607.865} C_VEL
LIN {X 0,Y 565.845,Z 633.936,A -85,B 0,C 180,E1 -2608.577,E2 -2608.577} C_VEL
LIN {X 0,Y 565.839,Z 634.71,A -85,B 0,C 180,E1 -2609.289,E2 -2609.289} C_VEL
LIN {X 0,Y 565.836,Z 635,A -85,B 0,C 180,E1 -2610,E2 -2610} C_VEL
LIN {X 0,Y 565.839,Z 634.71,A -85,B 0,C 180,E1 -2610.712,E2 -2610.712} C_VEL
LIN {X 0,Y 565.845,Z 633.934,A -85,B 0,C 180,E1 -2611.424,E2 -2611.424} C_VEL
LIN {X 0,Y 565.84,Z 632.68,A -85,B 0,C 180,E1 -2612.136,E2 -2612.136} C_VEL
LIN {X 0,Y 565.916,Z 629.787,A -85,B 0,C 180,E1 -2613.204,E2 -2613.204} C_VEL
LIN {X 0,Y 565.934,Z 627.146,A -85,B 0,C 180,E1 -2613.917,E2 -2613.917} C_VEL
LIN {X 0,Y 565.913,Z 621.984,A -85,B 0,C 180,E1 -2614.987,E2 -2614.987} C_VEL
LIN {X 0,Y 566.082,Z 615.184,A -85,B 0,C 180,E1 -2616.058,E2 -2616.058} C_VEL
LIN {X 0,Y 566.092,Z 608.175,A -85,B 0,C 180,E1 -2616.907,E2 -2616.907} C_VEL
LIN {X 0,Y 566.146,Z 600.403,A -85,B 0,C 180,E1 -2617.669,E2 -2617.669} C_VEL
LIN {X 0,Y 566.255,Z 592.54,A -85,B 0,C 180,E1 -2618.296,E2 -2618.296} C_VEL
LIN {X 0,Y 566.353,Z 582.725,A -85,B 0,C 180,E1 -2618.924,E2 -2618.924} C_VEL
LIN {X 0,Y 566.428,Z 571.293,A -85,B 0,C 180,E1 -2619.463,E2 -2619.463} C_VEL
LIN {X 0,Y 566.519,Z 561.233,A -85,B 0,C 180,E1 -2619.799,E2 -2619.799} C_VEL
LIN {X 0,Y 566.052,Z 554.367,A -85,B 0,C 180,E1 -2619.977,E2 -2619.977} C_VEL
LIN {X 0,Y 565.955,Z 553.301,A -85,B 0,C 180,E1 -2620.012,E2 -2620.012} C_VEL
LIN {X 0,Y 566.009,Z 544.36,A -85,B 0,C 180,E1 -2622.55,E2 -2622.55} C_VEL
LIN {X 0,Y 566.077,Z 534.141,A -85,B 0,C 180,E1 -2625.482,E2 -2625.482} C_VEL
LIN {X 0,Y 566.16,Z 523.922,A -85,B 0,C 180,E1 -2628.454,E2 -2628.454} C_VEL
LIN {X 0,Y 566.23,Z 513.882,A -85,B 0,C 180,E1 -2631.426,E2 -2631.426} C_VEL
LIN {X 0,Y 566.301,Z 504.664,A -85,B 0,C 180,E1 -2634.176,E2 -2634.176} C_VEL
LIN {X 0,Y 566.416,Z 495.314,A -85,B 0,C 180,E1 -2636.976,E2 -2636.976} C_VEL
LIN {X 0,Y 566.512,Z 486.475,A -85,B 0,C 180,E1 -2639.751,E2 -2639.751} C_VEL
LIN {X 0,Y 566.66,Z 479.087,A -85,B 0,C 180,E1 -2642.23,E2 -2642.23} C_VEL
LIN {X 0,Y 566.268,Z 474.765,A -85,B 0,C 180,E1 -2643.849,E2 -2643.849} C_VEL
LIN {X 0,Y 566.21,Z 474.769,A -85,B 0,C 180,E1 -2646.57,E2 -2646.57} C_VEL
LIN {X 0,Y 566.214,Z 474.768,A -85,B 0,C 180,E1 -2649.686,E2 -2649.686} C_VEL
LIN {X 0,Y 566.191,Z 474.772,A -85,B 0,C 180,E1 -2652.09,E2 -2652.09} C_VEL
LIN {X 0,Y 566.177,Z 474.776,A -85,B 0,C 180,E1 -2655.036,E2 -2655.036} C_VEL
LIN {X 0,Y 566.221,Z 474.771,A -85,B 0,C 180,E1 -2658.136,E2 -2658.136} C_VEL
LIN {X 0,Y 566.218,Z 474.766,A -85,B 0,C 180,E1 -2660.727,E2 -2660.727} C_VEL
LIN {X 0,Y 566.187,Z 474.77,A -85,B 0,C 180,E1 -2663.788,E2 -2663.788} C_VEL
LIN {X 0,Y 566.215,Z 474.772,A -85,B 0,C 180,E1 -2666.266,E2 -2666.266} C_VEL
LIN {X 0,Y 566.163,Z 474.778,A -85,B 0,C 180,E1 -2667.739,E2 -2667.739} C_VEL
LIN {X 0,Y 566.094,Z 475.2,A -85,B 0,C 180,E1 -2668.572,E2 -2668.572} C_VEL
LIN {X 0,Y 566.058,Z 478.524,A -85,B 0,C 180,E1 -2671.039,E2 -2671.039} C_VEL
LIN {X 0,Y 566.018,Z 481.773,A -85,B 0,C 180,E1 -2673.449,E2 -2673.449} C_VEL
LIN {X 0,Y 565.939,Z 485.981,A -85,B 0,C 180,E1 -2676.585,E2 -2676.585} C_VEL
LIN {X 0,Y 565.921,Z 489.296,A -85,B 0,C 180,E1 -2678.891,E2 -2678.891} C_VEL
LIN {X 0,Y 565.91,Z 492.742,A -85,B 0,C 180,E1 -2681.162,E2 -2681.162} C_VEL
LIN {X 0,Y 565.876,Z 497.337,A -85,B 0,C 180,E1 -2684.143,E2 -2684.143} C_VEL
LIN {X 0,Y 565.896,Z 500.784,A -85,B 0,C 180,E1 -2686.352,E2 -2686.352} C_VEL
LIN {X 0,Y 565.889,Z 505.379,A -85,B 0,C 180,E1 -2689.264,E2 -2689.264} C_VEL
LIN {X 0,Y 565.885,Z 506.708,A -85,B 0,C 180,E1 -2690.1,E2 -2690.1} C_VEL
LIN {X 0,Y 566.502,Z 513.741,A -85,B 0,C 180,E1 -2690.314,E2 -2690.314} C_VEL
LIN {X 0,Y 566.41,Z 524.592,A -85,B 0,C 180,E1 -2690.717,E2 -2690.717} C_VEL
LIN {X 0,Y 566.312,Z 534.981,A -85,B 0,C 180,E1 -2691.256,E2 -2691.256} C_VEL
LIN {X 0,Y 566.204,Z 543.159,A -85,B 0,C 180,E1 -2691.793,E2 -2691.793} C_VEL
LIN {X 0,Y 566.155,Z 550.913,A -85,B 0,C 180,E1 -2692.421,E2 -2692.421} C_VEL
LIN {X 0,Y 566.097,Z 557.71,A -85,B 0,C 180,E1 -2693.089,E2 -2693.089} C_VEL
LIN {X 0,Y 566.083,Z 564.837,A -85,B 0,C 180,E1 -2693.942,E2 -2693.942} C_VEL
LIN {X 0,Y 565.912,Z 571.745,A -85,B 0,C 180,E1 -2695.013,E2 -2695.013} C_VEL
LIN {X 0,Y 565.963,Z 575.44,A -85,B 0,C 180,E1 -2695.727,E2 -2695.727} C_VEL
LIN {X 0,Y 565.953,Z 578.454,A -85,B 0,C 180,E1 -2696.44,E2 -2696.44} C_VEL
LIN {X 0,Y 565.882,Z 580.789,A -85,B 0,C 180,E1 -2697.153,E2 -2697.153} C_VEL
LIN {X 0,Y 565.838,Z 582.58,A -85,B 0,C 180,E1 -2697.865,E2 -2697.865} C_VEL
LIN {X 0,Y 565.846,Z 583.874,A -85,B 0,C 180,E1 -2698.577,E2 -2698.577} C_VEL
LIN {X 0,Y 565.838,Z 584.69,A -85,B 0,C 180,E1 -2699.288,E2 -2699.288} C_VEL
LIN {X 0,Y 565.835,Z 584.996,A -85,B 0,C 180,E1 -2700,E2 -2700} C_VEL
LIN {X 0,Y 565.84,Z 584.73,A -85,B 0,C 180,E1 -2700.712,E2 -2700.712} C_VEL
LIN {X 0,Y 565.845,Z 583.996,A -85,B 0,C 180,E1 -2701.423,E2 -2701.423} C_VEL
LIN {X 0,Y 565.84,Z 582.782,A -85,B 0,C 180,E1 -2702.135,E2 -2702.135} C_VEL
LIN {X 0,Y 565.904,Z 579.933,A -85,B 0,C 180,E1 -2703.204,E2 -2703.204} C_VEL
LIN {X 0,Y 565.936,Z 577.339,A -85,B 0,C 180,E1 -2703.916,E2 -2703.916} C_VEL
LIN {X 0,Y 565.964,Z 574.14,A -85,B 0,C 180,E1 -2704.63,E2 -2704.63} C_VEL
LIN {X 0,Y 565.987,Z 569.079,A -85,B 0,C 180,E1 -2705.522,E2 -2705.522} C_VEL
LIN {X 0,Y 566.077,Z 564.135,A -85,B 0,C 180,E1 -2706.237,E2 -2706.237} C_VEL
LIN {X 0,Y 566.084,Z 558.162,A -85,B 0,C 180,E1 -2706.953,E2 -2706.953} C_VEL
LIN {X 0,Y 566.164,Z 549.893,A -85,B 0,C 180,E1 -2707.758,E2 -2707.758} C_VEL
LIN {X 0,Y 566.268,Z 541.928,A -85,B 0,C 180,E1 -2708.385,E2 -2708.385} C_VEL
LIN {X 0,Y 566.333,Z 531.952,A -85,B 0,C 180,E1 -2709.014,E2 -2709.014} C_VEL
LIN {X 0,Y 566.465,Z 521.298,A -85,B 0,C 180,E1 -2709.507,E2 -2709.507} C_VEL
LIN {X 0,Y 566.443,Z 511.238,A -85,B 0,C 180,E1 -2709.845,E2 -2709.845} C_VEL
LIN {X 0,Y 565.872,Z 506.519,A -85,B 0,C 180,E1 -2709.991,E2 -2709.991} C_VEL
LIN {X 0,Y 565.895,Z 502.813,A -85,B 0,C 180,E1 -2712.188,E2 -2712.188} C_VEL
LIN {X 0,Y 565.908,Z 497.922,A -85,B 0,C 180,E1 -2715.118,E2 -2715.118} C_VEL
LIN {X 0,Y 565.894,Z 493.031,A -85,B 0,C 180,E1 -2718.088,E2 -2718.088} C_VEL
LIN {X 0,Y 565.901,Z 489.363,A -85,B 0,C 180,E1 -2720.349,E2 -2720.349} C_VEL
LIN {X 0,Y 565.947,Z 484.793,A -85,B 0,C 180,E1 -2723.228,E2 -2723.228} C_VEL
LIN {X 0,Y 565.934,Z 483.727,A -85,B 0,C 180,E1 -2723.918,E2 -2723.918} C_VEL
LIN {X 0,Y 565.285,Z 482.915,A -85,B 0,C 180,E1 -2724.506,E2 -2724.506} C_VEL
LIN {X 0,Y 562.468,Z 481.792,A -85,B 0,C 180,E1 -2725.463,E2 -2725.463} C_VEL
LIN {X 0,Y 560.083,Z 480.823,A -85,B 0,C 180,E1 -2726.234,E2 -2726.234} C_VEL
LIN {X 0,Y 559.059,Z 479.984,A -85,B 0,C 180,E1 -2726.827,E2 -2726.827} C_VEL
LIN {X 0,Y 558.976,Z 479.68,A -85,B 0,C 180,E1 -2727.027,E2 -2727.027} C_VEL
LIN {X 0,Y 558.988,Z 479.385,A -85,B 0,C 180,E1 -2727.316,E2 -2727.316} C_VEL
LIN {X 0,Y 559.015,Z 485.782,A -85,B 0,C 180,E1 -2729.833,E2 -2729.833} C_VEL
LIN {X 0,Y 559.049,Z 492.681,A -85,B 0,C 180,E1 -2732.722,E2 -2732.722} C_VEL
LIN {X 0,Y 558.977,Z 500.241,A -85,B 0,C 180,E1 -2735.778,E2 -2735.778} C_VEL
LIN {X 0,Y 558.896,Z 507.412,A -85,B 0,C 180,E1 -2738.772,E2 -2738.772} C_VEL
LIN {X 0,Y 558.861,Z 512.857,A -85,B 0,C 180,E1 -2741.015,E2 -2741.015} C_VEL
LIN {X 0,Y 558.869,Z 519.597,A -85,B 0,C 180,E1 -2743.761,E2 -2743.761} C_VEL
LIN {X 0,Y 558.845,Z 525.028,A -85,B 0,C 180,E1 -2745.951,E2 -2745.951} C_VEL
LIN {X 0,Y 559.513,Z 532.768,A -85,B 0,C 180,E1 -2746.165,E2 -2746.165} C_VEL
LIN {X 0,Y 559.43,Z 544.043,A -85,B 0,C 180,E1 -2746.574,E2 -2746.574} C_VEL
LIN {X 0,Y 559.283,Z 555.057,A -85,B 0,C 180,E1 -2747.145,E2 -2747.145} C_VEL
LIN {X 0,Y 559.205,Z 564.111,A -85,B 0,C 180,E1 -2747.757,E2 -2747.757} C_VEL
LIN {X 0,Y 559.092,Z 572.053,A -85,B 0,C 180,E1 -2748.426,E2 -2748.426} C_VEL
LIN {X 0,Y 558.949,Z 580.261,A -85,B 0,C 180,E1 -2749.288,E2 -2749.288} C_VEL
LIN {X 0,Y 558.942,Z 586.574,A -85,B 0,C 180,E1 -2750.114,E2 -2750.114} C_VEL
LIN {X 0,Y 558.883,Z 592.274,A -85,B 0,C 180,E1 -2751.041,E2 -2751.041} C_VEL
LIN {X 0,Y 558.85,Z 596.685,A -85,B 0,C 180,E1 -2751.959,E2 -2751.959} C_VEL
LIN {X 0,Y 558.801,Z 600.024,A -85,B 0,C 180,E1 -2752.865,E2 -2752.865} C_VEL
LIN {X 0,Y 558.759,Z 602.433,A -85,B 0,C 180,E1 -2753.76,E2 -2753.76} C_VEL
LIN {X 0,Y 558.757,Z 604.26,A -85,B 0,C 180,E1 -2754.842,E2 -2754.842} C_VEL
LIN {X 0,Y 558.759,Z 604.991,A -85,B 0,C 180,E1 -2756.113,E2 -2756.113} C_VEL
LIN {X 0,Y 558.755,Z 604.021,A -85,B 0,C 180,E1 -2757.429,E2 -2757.429} C_VEL
LIN {X 0,Y 558.779,Z 602.915,A -85,B 0,C 180,E1 -2758.112,E2 -2758.112} C_VEL
LIN {X 0,Y 558.8,Z 600.87,A -85,B 0,C 180,E1 -2758.958,E2 -2758.958} C_VEL
LIN {X 0,Y 558.825,Z 598.066,A -85,B 0,C 180,E1 -2759.797,E2 -2759.797} C_VEL
LIN {X 0,Y 558.871,Z 593.401,A -85,B 0,C 180,E1 -2760.837,E2 -2760.837} C_VEL
LIN {X 0,Y 558.906,Z 587.642,A -85,B 0,C 180,E1 -2761.821,E2 -2761.821} C_VEL
LIN {X 0,Y 559.002,Z 581.269,A -85,B 0,C 180,E1 -2762.684,E2 -2762.684} C_VEL
LIN {X 0,Y 559.037,Z 573.831,A -85,B 0,C 180,E1 -2763.494,E2 -2763.494} C_VEL
LIN {X 0,Y 559.156,Z 565.781,A -85,B 0,C 180,E1 -2764.202,E2 -2764.202} C_VEL
LIN {X 0,Y 559.274,Z 557.466,A -85,B 0,C 180,E1 -2764.793,E2 -2764.793} C_VEL
LIN {X 0,Y 559.33,Z 548.445,A -85,B 0,C 180,E1 -2765.305,E2 -2765.305} C_VEL
LIN {X 0,Y 559.443,Z 539.268,A -85,B 0,C 180,E1 -2765.705,E2 -2765.705} C_VEL
LIN {X 0,Y 559.314,Z 529.524,A -85,B 0,C 180,E1 -2766.02,E2 -2766.02} C_VEL
LIN {X 0,Y 558.823,Z 525.266,A -85,B 0,C 180,E1 -2766.145,E2 -2766.145} C_VEL
LIN {X 0,Y 558.823,Z 519.529,A -85,B 0,C 180,E1 -2768.61,E2 -2768.61} C_VEL
LIN {X 0,Y 558.875,Z 514.206,A -85,B 0,C 180,E1 -2770.915,E2 -2770.915} C_VEL
LIN {X 0,Y 558.889,Z 507.315,A -85,B 0,C 180,E1 -2773.939,E2 -2773.939} C_VEL
LIN {X 0,Y 558.96,Z 502.281,A -85,B 0,C 180,E1 -2776.178,E2 -2776.178} C_VEL
LIN {X 0,Y 559,Z 495.651,A -85,B 0,C 180,E1 -2779.129,E2 -2779.129} C_VEL
LIN {X 0,Y 558.987,Z 488.949,A -85,B 0,C 180,E1 -2782.05,E2 -2782.05} C_VEL
LIN {X 0,Y 559.07,Z 482.235,A -85,B 0,C 180,E1 -2784.951,E2 -2784.951} C_VEL
LIN {X 0,Y 559,Z 475.67,A -85,B 0,C 180,E1 -2787.838,E2 -2787.838} C_VEL
LIN {X 0,Y 559.266,Z 475.634,A -85,B 0,C 180,E1 -2790,E2 -2790} C_VEL
LIN {X 0,Y 559.239,Z 475.64,A -85,B 0,C 180,E1 -2792.881,E2 -2792.881} C_VEL
LIN {X 0,Y 559.236,Z 475.638,A -85,B 0,C 180,E1 -2795.77,E2 -2795.77} C_VEL
LIN {X 0,Y 559.189,Z 475.646,A -85,B 0,C 180,E1 -2798.674,E2 -2798.674} C_VEL
LIN {X 0,Y 559.207,Z 475.641,A -85,B 0,C 180,E1 -2801.6,E2 -2801.6} C_VEL
LIN {X 0,Y 559.201,Z 475.644,A -85,B 0,C 180,E1 -2804.595,E2 -2804.595} C_VEL
LIN {X 0,Y 559.164,Z 475.647,A -85,B 0,C 180,E1 -2807.556,E2 -2807.556} C_VEL
LIN {X 0,Y 559.174,Z 475.646,A -85,B 0,C 180,E1 -2809.837,E2 -2809.837} C_VEL
LIN {X 0,Y 559.142,Z 475.65,A -85,B 0,C 180,E1 -2812.152,E2 -2812.152} C_VEL
LIN {X 0,Y 559.181,Z 475.646,A -85,B 0,C 180,E1 -2815.187,E2 -2815.187} C_VEL
LIN {X 0,Y 559.192,Z 475.646,A -85,B 0,C 180,E1 -2817.711,E2 -2817.711} C_VEL
LIN {X 0,Y 559.17,Z 475.648,A -85,B 0,C 180,E1 -2820.181,E2 -2820.181} C_VEL
LIN {X 0,Y 559.176,Z 475.646,A -85,B 0,C 180,E1 -2822.713,E2 -2822.713} C_VEL
LIN {X 0,Y 559.158,Z 475.647,A -85,B 0,C 180,E1 -2825.321,E2 -2825.321} C_VEL
LIN {X 0,Y 559.136,Z 475.651,A -85,B 0,C 180,E1 -2828.017,E2 -2828.017} C_VEL
LIN {X 0,Y 559.172,Z 475.647,A -85,B 0,C 180,E1 -2830.81,E2 -2830.81} C_VEL
LIN {X 0,Y 559.162,Z 475.647,A -85,B 0,C 180,E1 -2833.731,E2 -2833.731} C_VEL
LIN {X 0,Y 559.167,Z 475.647,A -85,B 0,C 180,E1 -2836.801,E2 -2836.801} C_VEL
LIN {X 0,Y 559.179,Z 475.646,A -85,B 0,C 180,E1 -2839.19,E2 -2839.19} C_VEL
LIN {X 0,Y 559.134,Z 475.651,A -85,B 0,C 180,E1 -2841.982,E2 -2841.982} C_VEL
LIN {X 0,Y 559.131,Z 475.654,A -85,B 0,C 180,E1 -2844.787,E2 -2844.787} C_VEL
LIN {X 0,Y 559.174,Z 475.648,A -85,B 0,C 180,E1 -2847.361,E2 -2847.361} C_VEL
LIN {X 0,Y 559.148,Z 475.649,A -85,B 0,C 180,E1 -2850.142,E2 -2850.142} C_VEL
LIN {X 0,Y 559.181,Z 475.647,A -85,B 0,C 180,E1 -2853.17,E2 -2853.17} C_VEL
LIN {X 0,Y 559.155,Z 475.65,A -85,B 0,C 180,E1 -2855.495,E2 -2855.495} C_VEL
LIN {X 0,Y 559.177,Z 475.645,A -85,B 0,C 180,E1 -2858.624,E2 -2858.624} C_VEL
LIN {X 0,Y 559.168,Z 475.645,A -85,B 0,C 180,E1 -2860.926,E2 -2860.926} C_VEL
LIN {X 0,Y 559.168,Z 475.648,A -85,B 0,C 180,E1 -2863.948,E2 -2863.948} C_VEL
LIN {X 0,Y 559.173,Z 475.648,A -85,B 0,C 180,E1 -2866.184,E2 -2866.184} C_VEL
LIN {X 0,Y 559.193,Z 475.643,A -85,B 0,C 180,E1 -2869.133,E2 -2869.133} C_VEL
LIN {X 0,Y 559.205,Z 475.645,A -85,B 0,C 180,E1 -2872.054,E2 -2872.054} C_VEL
LIN {X 0,Y 559.253,Z 475.635,A -85,B 0,C 180,E1 -2874.953,E2 -2874.953} C_VEL
LIN {X 0,Y 559.254,Z 475.638,A -85,B 0,C 180,E1 -2877.839,E2 -2877.839} C_VEL
LIN {X 0,Y 559.273,Z 475.633,A -85,B 0,C 180,E1 -2880.72,E2 -2880.72} C_VEL
LIN {X 0,Y 559.242,Z 475.639,A -85,B 0,C 180,E1 -2882.881,E2 -2882.881} C_VEL
LIN {X 0,Y 559.231,Z 475.639,A -85,B 0,C 180,E1 -2885.77,E2 -2885.77} C_VEL
LIN {X 0,Y 559.191,Z 475.646,A -85,B 0,C 180,E1 -2888.674,E2 -2888.674} C_VEL
LIN {X 0,Y 559.203,Z 475.642,A -85,B 0,C 180,E1 -2891.6,E2 -2891.6} C_VEL
LIN {X 0,Y 559.197,Z 475.645,A -85,B 0,C 180,E1 -2894.596,E2 -2894.596} C_VEL
LIN {X 0,Y 559.163,Z 475.647,A -85,B 0,C 180,E1 -2897.557,E2 -2897.557} C_VEL
LIN {X 0,Y 559.17,Z 475.646,A -85,B 0,C 180,E1 -2899.837,E2 -2899.837} C_VEL
LIN {X 0,Y 559.141,Z 475.649,A -85,B 0,C 180,E1 -2902.153,E2 -2902.153} C_VEL
LIN {X 0,Y 559.177,Z 475.648,A -85,B 0,C 180,E1 -2905.187,E2 -2905.187} C_VEL
LIN {X 0,Y 559.186,Z 475.645,A -85,B 0,C 180,E1 -2907.712,E2 -2907.712} C_VEL
LIN {X 0,Y 559.167,Z 475.646,A -85,B 0,C 180,E1 -2910.182,E2 -2910.182} C_VEL
LIN {X 0,Y 559.174,Z 475.645,A -85,B 0,C 180,E1 -2912.714,E2 -2912.714} C_VEL
LIN {X 0,Y 559.156,Z 475.648,A -85,B 0,C 180,E1 -2915.322,E2 -2915.322} C_VEL
LIN {X 0,Y 559.132,Z 475.653,A -85,B 0,C 180,E1 -2918.018,E2 -2918.018} C_VEL
LIN {X 0,Y 559.189,Z 475.644,A -85,B 0,C 180,E1 -2921.055,E2 -2921.055} C_VEL
LIN {X 0,Y 559.163,Z 475.648,A -85,B 0,C 180,E1 -2923.732,E2 -2923.732} C_VEL
LIN {X 0,Y 559.145,Z 475.649,A -85,B 0,C 180,E1 -2926.804,E2 -2926.804} C_VEL
LIN {X 0,Y 559.176,Z 475.646,A -85,B 0,C 180,E1 -2929.19,E2 -2929.19} C_VEL
LIN {X 0,Y 559.134,Z 475.651,A -85,B 0,C 180,E1 -2931.983,E2 -2931.983} C_VEL
LIN {X 0,Y 559.16,Z 475.65,A -85,B 0,C 180,E1 -2934.783,E2 -2934.783} C_VEL
LIN {X 0,Y 559.231,Z 475.832,A -85,B 0,C 180,E1 -2937.823,E2 -2937.823} C_VEL
LIN {X 0,Y 559.68,Z 479.518,A -85,B 0,C 180,E1 -2939.013,E2 -2939.013} C_VEL
LIN {X 0,Y 559.563,Z 487.725,A -85,B 0,C 180,E1 -2941.544,E2 -2941.544} C_VEL
LIN {X 0,Y 559.433,Z 497.13,A -85,B 0,C 180,E1 -2944.316,E2 -2944.316} C_VEL
LIN {X 0,Y 559.295,Z 506.735,A -85,B 0,C 180,E1 -2947.075,E2 -2947.075} C_VEL
LIN {X 0,Y 559.222,Z 516.288,A -85,B 0,C 180,E1 -2949.782,E2 -2949.782} C_VEL
LIN {X 0,Y 559.119,Z 527.106,A -85,B 0,C 180,E1 -2952.805,E2 -2952.805} C_VEL
LIN {X 0,Y 558.994,Z 538.09,A -85,B 0,C 180,E1 -2955.825,E2 -2955.825} C_VEL
LIN {X 0,Y 558.972,Z 548.761,A -85,B 0,C 180,E1 -2958.725,E2 -2958.725} C_VEL
LIN {X 0,Y 558.915,Z 552.978,A -85,B 0,C 180,E1 -2959.861,E2 -2959.861} C_VEL
LIN {X 0,Y 559.502,Z 560.426,A -85,B 0,C 180,E1 -2960.055,E2 -2960.055} C_VEL
LIN {X 0,Y 559.464,Z 568.899,A -85,B 0,C 180,E1 -2960.328,E2 -2960.328} C_VEL
LIN {X 0,Y 559.39,Z 577.405,A -85,B 0,C 180,E1 -2960.691,E2 -2960.691} C_VEL
LIN {X 0,Y 559.299,Z 585.735,A -85,B 0,C 180,E1 -2961.146,E2 -2961.146} C_VEL
LIN {X 0,Y 559.194,Z 593.774,A -85,B 0,C 180,E1 -2961.69,E2 -2961.69} C_VEL
LIN {X 0,Y 559.094,Z 602.435,A -85,B 0,C 180,E1 -2962.416,E2 -2962.416} C_VEL
LIN {X 0,Y 558.983,Z 611.084,A -85,B 0,C 180,E1 -2963.34,E2 -2963.34} C_VEL
LIN {X 0,Y 558.969,Z 617.614,A -85,B 0,C 180,E1 -2964.228,E2 -2964.228} C_VEL
LIN {X 0,Y 558.827,Z 621.99,A -85,B 0,C 180,E1 -2964.95,E2 -2964.95} C_VEL
LIN {X 0,Y 558.858,Z 627.15,A -85,B 0,C 180,E1 -2966.034,E2 -2966.034} C_VEL
LIN {X 0,Y 558.805,Z 630.936,A -85,B 0,C 180,E1 -2967.117,E2 -2967.117} C_VEL
LIN {X 0,Y 558.746,Z 632.683,A -85,B 0,C 180,E1 -2967.838,E2 -2967.838} C_VEL
LIN {X 0,Y 558.744,Z 633.935,A -85,B 0,C 180,E1 -2968.559,E2 -2968.559} C_VEL
LIN {X 0,Y 558.739,Z 634.71,A -85,B 0,C 180,E1 -2969.28,E2 -2969.28} C_VEL
LIN {X 0,Y 558.737,Z 635,A -85,B 0,C 180,E1 -2970,E2 -2970} C_VEL
LIN {X 0,Y 558.739,Z 634.709,A -85,B 0,C 180,E1 -2970.721,E2 -2970.721} C_VEL
LIN {X 0,Y 558.744,Z 633.933,A -85,B 0,C 180,E1 -2971.442,E2 -2971.442} C_VEL
LIN {X 0,Y 558.746,Z 632.681,A -85,B 0,C 180,E1 -2972.163,E2 -2972.163} C_VEL
LIN {X 0,Y 558.841,Z 629.786,A -85,B 0,C 180,E1 -2973.245,E2 -2973.245} C_VEL
LIN {X 0,Y 558.851,Z 627.147,A -85,B 0,C 180,E1 -2973.966,E2 -2973.966} C_VEL
LIN {X 0,Y 558.827,Z 621.984,A -85,B 0,C 180,E1 -2975.051,E2 -2975.051} C_VEL
LIN {X 0,Y 559.018,Z 615.183,A -85,B 0,C 180,E1 -2976.135,E2 -2976.135} C_VEL
LIN {X 0,Y 559.036,Z 607.741,A -85,B 0,C 180,E1 -2977.041,E2 -2977.041} C_VEL
LIN {X 0,Y 559.12,Z 600.401,A -85,B 0,C 180,E1 -2977.766,E2 -2977.766} C_VEL
LIN {X 0,Y 559.24,Z 592.538,A -85,B 0,C 180,E1 -2978.401,E2 -2978.401} C_VEL
LIN {X 0,Y 559.317,Z 582.723,A -85,B 0,C 180,E1 -2979.037,E2 -2979.037} C_VEL
LIN {X 0,Y 559.437,Z 571.294,A -85,B 0,C 180,E1 -2979.582,E2 -2979.582} C_VEL
LIN {X 0,Y 559.527,Z 561.233,A -85,B 0,C 180,E1 -2979.923,E2 -2979.923} C_VEL
LIN {X 0,Y 558.996,Z 554.366,A -85,B 0,C 180,E1 -2980.104,E2 -2980.104} C_VEL
LIN {X 0,Y 558.895,Z 553.301,A -85,B 0,C 180,E1 -2980.14,E2 -2980.14} C_VEL
LIN {X 0,Y 558.937,Z 544.36,A -85,B 0,C 180,E1 -2982.712,E2 -2982.712} C_VEL
LIN {X 0,Y 559.021,Z 535.418,A -85,B 0,C 180,E1 -2985.309,E2 -2985.309} C_VEL
LIN {X 0,Y 559.11,Z 525.2,A -85,B 0,C 180,E1 -2988.316,E2 -2988.316} C_VEL
LIN {X 0,Y 559.175,Z 516.258,A -85,B 0,C 180,E1 -2990.99,E2 -2990.99} C_VEL
LIN {X 0,Y 559.291,Z 507.068,A -85,B 0,C 180,E1 -2993.71,E2 -2993.71} C_VEL
LIN {X 0,Y 559.366,Z 497.896,A -85,B 0,C 180,E1 -2996.479,E2 -2996.479} C_VEL
LIN {X 0,Y 559.484,Z 488.907,A -85,B 0,C 180,E1 -2999.334,E2 -2999.334} C_VEL
LIN {X 0,Y 559.674,Z 481.53,A -85,B 0,C 180,E1 -3001.831,E2 -3001.831} C_VEL
LIN {X 0,Y 559.583,Z 478.031,A -85,B 0,C 180,E1 -3003.116,E2 -3003.116} C_VEL
LIN {X 0,Y 559.221,Z 475.643,A -85,B 0,C 180,E1 -3004.065,E2 -3004.065} C_VEL
LIN {X 0,Y 559.146,Z 475.652,A -85,B 0,C 180,E1 -3007.108,E2 -3007.108} C_VEL
LIN {X 0,Y 559.167,Z 475.648,A -85,B 0,C 180,E1 -3009.943,E2 -3009.943} C_VEL
LIN {X 0,Y 559.16,Z 475.645,A -85,B 0,C 180,E1 -3012.744,E2 -3012.744} C_VEL
LIN {X 0,Y 559.158,Z 475.645,A -85,B 0,C 180,E1 -3015.761,E2 -3015.761} C_VEL
LIN {X 0,Y 559.192,Z 475.646,A -85,B 0,C 180,E1 -3018.232,E2 -3018.232} C_VEL
LIN {X 0,Y 559.178,Z 475.647,A -85,B 0,C 180,E1 -3021.192,E2 -3021.192} C_VEL
LIN {X 0,Y 559.142,Z 475.648,A -85,B 0,C 180,E1 -3023.789,E2 -3023.789} C_VEL
LIN {X 0,Y 559.163,Z 475.649,A -85,B 0,C 180,E1 -3026.425,E2 -3026.425} C_VEL
LIN {X 0,Y 559.074,Z 475.661,A -85,B 0,C 180,E1 -3028.131,E2 -3028.131} C_VEL
LIN {X 0,Y 559.02,Z 478.128,A -85,B 0,C 180,E1 -3030.166,E2 -3030.166} C_VEL
LIN {X 0,Y 558.955,Z 482.035,A -85,B 0,C 180,E1 -3033.087,E2 -3033.087} C_VEL
LIN {X 0,Y 558.871,Z 485.176,A -85,B 0,C 180,E1 -3035.482,E2 -3035.482} C_VEL
LIN {X 0,Y 558.844,Z 489.319,A -85,B 0,C 180,E1 -3038.533,E2 -3038.533} C_VEL
LIN {X 0,Y 558.837,Z 492.743,A -85,B 0,C 180,E1 -3040.915,E2 -3040.915} C_VEL
LIN {X 0,Y 558.785,Z 497.338,A -85,B 0,C 180,E1 -3043.937,E2 -3043.937} C_VEL
LIN {X 0,Y 558.799,Z 500.784,A -85,B 0,C 180,E1 -3046.175,E2 -3046.175} C_VEL
LIN {X 0,Y 558.81,Z 505.38,A -85,B 0,C 180,E1 -3049.126,E2 -3049.126} C_VEL
LIN {X 0,Y 558.801,Z 506.708,A -85,B 0,C 180,E1 -3049.973,E2 -3049.973} C_VEL
LIN {X 0,Y 559.514,Z 513.763,A -85,B 0,C 180,E1 -3050.191,E2 -3050.191} C_VEL
LIN {X 0,Y 559.412,Z 524.602,A -85,B 0,C 180,E1 -3050.6,E2 -3050.6} C_VEL
LIN {X 0,Y 559.297,Z 534.989,A -85,B 0,C 180,E1 -3051.145,E2 -3051.145} C_VEL
LIN {X 0,Y 559.181,Z 543.164,A -85,B 0,C 180,E1 -3051.69,E2 -3051.69} C_VEL
LIN {X 0,Y 559.106,Z 550.92,A -85,B 0,C 180,E1 -3052.325,E2 -3052.325} C_VEL
LIN {X 0,Y 559.019,Z 559.024,A -85,B 0,C 180,E1 -3053.141,E2 -3053.141} C_VEL
LIN {X 0,Y 559.005,Z 566.139,A -85,B 0,C 180,E1 -3054.047,E2 -3054.047} C_VEL
LIN {X 0,Y 558.826,Z 571.748,A -85,B 0,C 180,E1 -3054.95,E2 -3054.95} C_VEL
LIN {X 0,Y 558.896,Z 575.443,A -85,B 0,C 180,E1 -3055.673,E2 -3055.673} C_VEL
LIN {X 0,Y 558.842,Z 579.644,A -85,B 0,C 180,E1 -3056.756,E2 -3056.756} C_VEL
LIN {X 0,Y 558.744,Z 582.582,A -85,B 0,C 180,E1 -3057.838,E2 -3057.838} C_VEL
LIN {X 0,Y 558.745,Z 583.873,A -85,B 0,C 180,E1 -3058.559,E2 -3058.559} C_VEL
LIN {X 0,Y 558.738,Z 584.689,A -85,B 0,C 180,E1 -3059.279,E2 -3059.279} C_VEL
LIN {X 0,Y 558.736,Z 584.996,A -85,B 0,C 180,E1 -3060,E2 -3060} C_VEL
LIN {X 0,Y 558.74,Z 584.729,A -85,B 0,C 180,E1 -3060.721,E2 -3060.721} C_VEL
LIN {X 0,Y 558.744,Z 583.994,A -85,B 0,C 180,E1 -3061.442,E2 -3061.442} C_VEL
LIN {X 0,Y 558.746,Z 582.782,A -85,B 0,C 180,E1 -3062.163,E2 -3062.163} C_VEL
LIN {X 0,Y 558.829,Z 579.931,A -85,B 0,C 180,E1 -3063.244,E2 -3063.244} C_VEL
LIN {X 0,Y 558.853,Z 577.337,A -85,B 0,C 180,E1 -3063.966,E2 -3063.966} C_VEL
LIN {X 0,Y 558.814,Z 572.226,A -85,B 0,C 180,E1 -3065.051,E2 -3065.051} C_VEL
LIN {X 0,Y 559.003,Z 566.727,A -85,B 0,C 180,E1 -3065.954,E2 -3065.954} C_VEL
LIN {X 0,Y 559.027,Z 558.333,A -85,B 0,C 180,E1 -3067.023,E2 -3067.023} C_VEL
LIN {X 0,Y 559.119,Z 550.905,A -85,B 0,C 180,E1 -3067.766,E2 -3067.766} C_VEL
LIN {X 0,Y 559.222,Z 543.146,A -85,B 0,C 180,E1 -3068.401,E2 -3068.401} C_VEL
LIN {X 0,Y 559.345,Z 534.968,A -85,B 0,C 180,E1 -3068.945,E2 -3068.945} C_VEL
LIN {X 0,Y 559.403,Z 526.446,A -85,B 0,C 180,E1 -3069.4,E2 -3069.4} C_VEL
LIN {X 0,Y 559.499,Z 515.204,A -85,B 0,C 180,E1 -3069.855,E2 -3069.855} C_VEL
LIN {X 0,Y 558.991,Z 508.306,A -85,B 0,C 180,E1 -3070.058,E2 -3070.058} C_VEL
LIN {X 0,Y 558.791,Z 506.48,A -85,B 0,C 180,E1 -3070.142,E2 -3070.142} C_VEL
LIN {X 0,Y 558.797,Z 502.812,A -85,B 0,C 180,E1 -3072.346,E2 -3072.346} C_VEL
LIN {X 0,Y 558.823,Z 497.921,A -85,B 0,C 180,E1 -3075.314,E2 -3075.314} C_VEL
LIN {X 0,Y 558.795,Z 494.253,A -85,B 0,C 180,E1 -3077.569,E2 -3077.569} C_VEL
LIN {X 0,Y 558.835,Z 490.585,A -85,B 0,C 180,E1 -3079.85,E2 -3079.85} C_VEL
LIN {X 0,Y 558.847,Z 486.962,A -85,B 0,C 180,E1 -3082.165,E2 -3082.165} C_VEL
LIN {X 0,Y 558.874,Z 483.54,A -85,B 0,C 180,E1 -3084.518,E2 -3084.518} C_VEL
LIN {X 0,Y 558.976,Z 479.68,A -85,B 0,C 180,E1 -3087.027,E2 -3087.027} C_VEL
LIN {X 0,Y 558.655,Z 479.812,A -85,B 0,C 180,E1 -3087.426,E2 -3087.426} C_VEL
LIN {X 0,Y 556.748,Z 481.82,A -85,B 0,C 180,E1 -3088.195,E2 -3088.195} C_VEL
LIN {X 0,Y 553.105,Z 485.124,A -85,B 0,C 180,E1 -3089.324,E2 -3089.324} C_VEL
LIN {X 0,Y 552.044,Z 486.611,A -85,B 0,C 180,E1 -3089.913,E2 -3089.913} C_VEL
LIN {X 0,Y 551.947,Z 487.104,A -85,B 0,C 180,E1 -3090.113,E2 -3090.113} C_VEL
LIN {X 0,Y 551.969,Z 494.457,A -85,B 0,C 180,E1 -3093.196,E2 -3093.196} C_VEL
LIN {X 0,Y 551.892,Z 500.886,A -85,B 0,C 180,E1 -3095.858,E2 -3095.858} C_VEL
LIN {X 0,Y 551.814,Z 507.58,A -85,B 0,C 180,E1 -3098.614,E2 -3098.614} C_VEL
LIN {X 0,Y 551.788,Z 514.445,A -85,B 0,C 180,E1 -3101.476,E2 -3101.476} C_VEL
LIN {X 0,Y 551.772,Z 521.786,A -85,B 0,C 180,E1 -3104.497,E2 -3104.497} C_VEL
LIN {X 0,Y 551.783,Z 525.207,A -85,B 0,C 180,E1 -3105.824,E2 -3105.824} C_VEL
LIN {X 0,Y 552.524,Z 533.362,A -85,B 0,C 180,E1 -3106.057,E2 -3106.057} C_VEL
LIN {X 0,Y 552.422,Z 544.721,A -85,B 0,C 180,E1 -3106.482,E2 -3106.482} C_VEL
LIN {X 0,Y 552.257,Z 556.006,A -85,B 0,C 180,E1 -3107.09,E2 -3107.09} C_VEL
LIN {X 0,Y 552.139,Z 565.102,A -85,B 0,C 180,E1 -3107.73,E2 -3107.73} C_VEL
LIN {X 0,Y 552.034,Z 573.026,A -85,B 0,C 180,E1 -3108.424,E2 -3108.424} C_VEL
LIN {X 0,Y 551.898,Z 580.745,A -85,B 0,C 180,E1 -3109.259,E2 -3109.259} C_VEL
LIN {X 0,Y 551.869,Z 587.27,A -85,B 0,C 180,E1 -3110.139,E2 -3110.139} C_VEL
LIN {X 0,Y 551.777,Z 593.356,A -85,B 0,C 180,E1 -3111.182,E2 -3111.182} C_VEL
LIN {X 0,Y 551.753,Z 598.29,A -85,B 0,C 180,E1 -3112.309,E2 -3112.309} C_VEL
LIN {X 0,Y 551.685,Z 601.591,A -85,B 0,C 180,E1 -3113.376,E2 -3113.376} C_VEL
LIN {X 0,Y 551.656,Z 603.272,A -85,B 0,C 180,E1 -3114.124,E2 -3114.124} C_VEL
LIN {X 0,Y 551.657,Z 604.506,A -85,B 0,C 180,E1 -3115.02,E2 -3115.02} C_VEL
LIN {X 0,Y 551.677,Z 604.966,A -85,B 0,C 180,E1 -3115.907,E2 -3115.907} C_VEL
LIN {X 0,Y 551.669,Z 604.311,A -85,B 0,C 180,E1 -3117.226,E2 -3117.226} C_VEL
LIN {X 0,Y 551.735,Z 601.887,A -85,B 0,C 180,E1 -3118.589,E2 -3118.589} C_VEL
LIN {X 0,Y 551.725,Z 598.491,A -85,B 0,C 180,E1 -3119.722,E2 -3119.722} C_VEL
LIN {X 0,Y 551.787,Z 593.692,A -85,B 0,C 180,E1 -3120.844,E2 -3120.844} C_VEL
LIN {X 0,Y 551.83,Z 587.712,A -85,B 0,C 180,E1 -3121.886,E2 -3121.886} C_VEL
LIN {X 0,Y 551.93,Z 581.715,A -85,B 0,C 180,E1 -3122.715,E2 -3122.715} C_VEL
LIN {X 0,Y 551.975,Z 574.373,A -85,B 0,C 180,E1 -3123.536,E2 -3123.536} C_VEL
LIN {X 0,Y 552.114,Z 566.431,A -85,B 0,C 180,E1 -3124.253,E2 -3124.253} C_VEL
LIN {X 0,Y 552.239,Z 558.415,A -85,B 0,C 180,E1 -3124.843,E2 -3124.843} C_VEL
LIN {X 0,Y 552.31,Z 549.44,A -85,B 0,C 180,E1 -3125.371,E2 -3125.371} C_VEL
LIN {X 0,Y 552.452,Z 540.528,A -85,B 0,C 180,E1 -3125.778,E2 -3125.778} C_VEL
LIN {X 0,Y 552.458,Z 531.167,A -85,B 0,C 180,E1 -3126.098,E2 -3126.098} C_VEL
LIN {X 0,Y 551.715,Z 525.252,A -85,B 0,C 180,E1 -3126.283,E2 -3126.283} C_VEL
LIN {X 0,Y 551.73,Z 518.774,A -85,B 0,C 180,E1 -3129.104,E2 -3129.104} C_VEL
LIN {X 0,Y 551.77,Z 513.481,A -85,B 0,C 180,E1 -3131.432,E2 -3131.432} C_VEL
LIN {X 0,Y 551.808,Z 508.318,A -85,B 0,C 180,E1 -3133.728,E2 -3133.728} C_VEL
LIN {X 0,Y 551.877,Z 503.228,A -85,B 0,C 180,E1 -3135.997,E2 -3135.997} C_VEL
LIN {X 0,Y 551.95,Z 496.543,A -85,B 0,C 180,E1 -3138.989,E2 -3138.989} C_VEL
LIN {X 0,Y 551.927,Z 489.816,A -85,B 0,C 180,E1 -3141.948,E2 -3141.948} C_VEL
LIN {X 0,Y 552.015,Z 483.086,A -85,B 0,C 180,E1 -3144.887,E2 -3144.887} C_VEL
LIN {X 0,Y 551.926,Z 476.551,A -85,B 0,C 180,E1 -3147.719,E2 -3147.719} C_VEL
LIN {X 0,Y 552.245,Z 476.511,A -85,B 0,C 180,E1 -3149.27,E2 -3149.27} C_VEL
LIN {X 0,Y 552.228,Z 476.511,A -85,B 0,C 180,E1 -3152.188,E2 -3152.188} C_VEL
LIN {X 0,Y 552.232,Z 476.512,A -85,B 0,C 180,E1 -3155.111,E2 -3155.111} C_VEL
LIN {X 0,Y 552.16,Z 476.52,A -85,B 0,C 180,E1 -3158.048,E2 -3158.048} C_VEL
LIN {X 0,Y 552.177,Z 476.518,A -85,B 0,C 180,E1 -3161.466,E2 -3161.466} C_VEL
LIN {X 0,Y 552.159,Z 476.522,A -85,B 0,C 180,E1 -3164.682,E2 -3164.682} C_VEL
LIN {X 0,Y 552.115,Z 476.525,A -85,B 0,C 180,E1 -3167.788,E2 -3167.788} C_VEL
LIN {X 0,Y 552.133,Z 476.523,A -85,B 0,C 180,E1 -3170.101,E2 -3170.101} C_VEL
LIN {X 0,Y 552.096,Z 476.527,A -85,B 0,C 180,E1 -3172.45,E2 -3172.45} C_VEL
LIN {X 0,Y 552.158,Z 476.522,A -85,B 0,C 180,E1 -3175.35,E2 -3175.35} C_VEL
LIN {X 0,Y 552.125,Z 476.524,A -85,B 0,C 180,E1 -3178.097,E2 -3178.097} C_VEL
LIN {X 0,Y 552.116,Z 476.525,A -85,B 0,C 180,E1 -3180.608,E2 -3180.608} C_VEL
LIN {X 0,Y 552.124,Z 476.523,A -85,B 0,C 180,E1 -3183.185,E2 -3183.185} C_VEL
LIN {X 0,Y 552.114,Z 476.527,A -85,B 0,C 180,E1 -3185.841,E2 -3185.841} C_VEL
LIN {X 0,Y 552.125,Z 476.523,A -85,B 0,C 180,E1 -3189.062,E2 -3189.062} C_VEL
LIN {X 0,Y 552.127,Z 476.523,A -85,B 0,C 180,E1 -3191.445,E2 -3191.445} C_VEL
LIN {X 0,Y 552.096,Z 476.528,A -85,B 0,C 180,E1 -3194.532,E2 -3194.532} C_VEL
LIN {X 0,Y 552.13,Z 476.524,A -85,B 0,C 180,E1 -3197.584,E2 -3197.584} C_VEL
LIN {X 0,Y 552.134,Z 476.523,A -85,B 0,C 180,E1 -3200.473,E2 -3200.473} C_VEL
LIN {X 0,Y 552.104,Z 476.526,A -85,B 0,C 180,E1 -3203.317,E2 -3203.317} C_VEL
LIN {X 0,Y 552.126,Z 476.526,A -85,B 0,C 180,E1 -3205.939,E2 -3205.939} C_VEL
LIN {X 0,Y 552.117,Z 476.526,A -85,B 0,C 180,E1 -3208.54,E2 -3208.54} C_VEL
LIN {X 0,Y 552.124,Z 476.523,A -85,B 0,C 180,E1 -3211.437,E2 -3211.437} C_VEL
LIN {X 0,Y 552.136,Z 476.524,A -85,B 0,C 180,E1 -3214.356,E2 -3214.356} C_VEL
LIN {X 0,Y 552.108,Z 476.528,A -85,B 0,C 180,E1 -3216.758,E2 -3216.758} C_VEL
LIN {X 0,Y 552.126,Z 476.526,A -85,B 0,C 180,E1 -3219.12,E2 -3219.12} C_VEL
LIN {X 0,Y 552.125,Z 476.526,A -85,B 0,C 180,E1 -3221.444,E2 -3221.444} C_VEL
LIN {X 0,Y 552.118,Z 476.527,A -85,B 0,C 180,E1 -3223.737,E2 -3223.737} C_VEL
LIN {X 0,Y 552.136,Z 476.524,A -85,B 0,C 180,E1 -3226.004,E2 -3226.004} C_VEL
LIN {X 0,Y 552.16,Z 476.519,A -85,B 0,C 180,E1 -3228.993,E2 -3228.993} C_VEL
LIN {X 0,Y 552.159,Z 476.522,A -85,B 0,C 180,E1 -3231.951,E2 -3231.951} C_VEL
LIN {X 0,Y 552.227,Z 476.51,A -85,B 0,C 180,E1 -3234.889,E2 -3234.889} C_VEL
LIN {X 0,Y 552.225,Z 476.513,A -85,B 0,C 180,E1 -3237.812,E2 -3237.812} C_VEL
LIN {X 0,Y 552.242,Z 476.509,A -85,B 0,C 180,E1 -3240.729,E2 -3240.729} C_VEL
LIN {X 0,Y 552.208,Z 476.514,A -85,B 0,C 180,E1 -3242.918,E2 -3242.918} C_VEL
LIN {X 0,Y 552.201,Z 476.515,A -85,B 0,C 180,E1 -3245.844,E2 -3245.844} C_VEL
LIN {X 0,Y 552.161,Z 476.52,A -85,B 0,C 180,E1 -3248.786,E2 -3248.786} C_VEL
LIN {X 0,Y 552.161,Z 476.52,A -85,B 0,C 180,E1 -3251.75,E2 -3251.75} C_VEL
LIN {X 0,Y 552.135,Z 476.523,A -85,B 0,C 180,E1 -3254.748,E2 -3254.748} C_VEL
LIN {X 0,Y 552.114,Z 476.526,A -85,B 0,C 180,E1 -3257.788,E2 -3257.788} C_VEL
LIN {X 0,Y 552.129,Z 476.524,A -85,B 0,C 180,E1 -3260.101,E2 -3260.101} C_VEL
LIN {X 0,Y 552.095,Z 476.528,A -85,B 0,C 180,E1 -3262.451,E2 -3262.451} C_VEL
LIN {X 0,Y 552.153,Z 476.522,A -85,B 0,C 180,E1 -3265.351,E2 -3265.351} C_VEL
LIN {X 0,Y 552.121,Z 476.524,A -85,B 0,C 180,E1 -3268.098,E2 -3268.098} C_VEL
LIN {X 0,Y 552.113,Z 476.525,A -85,B 0,C 180,E1 -3270.609,E2 -3270.609} C_VEL
LIN {X 0,Y 552.121,Z 476.525,A -85,B 0,C 180,E1 -3273.185,E2 -3273.185} C_VEL
LIN {X 0,Y 552.112,Z 476.527,A -85,B 0,C 180,E1 -3275.842,E2 -3275.842} C_VEL
LIN {X 0,Y 552.12,Z 476.525,A -85,B 0,C 180,E1 -3279.062,E2 -3279.062} C_VEL
LIN {X 0,Y 552.139,Z 476.523,A -85,B 0,C 180,E1 -3281.444,E2 -3281.444} C_VEL
LIN {X 0,Y 552.095,Z 476.527,A -85,B 0,C 180,E1 -3284.532,E2 -3284.532} C_VEL
LIN {X 0,Y 552.129,Z 476.526,A -85,B 0,C 180,E1 -3287.585,E2 -3287.585} C_VEL
LIN {X 0,Y 552.134,Z 476.522,A -85,B 0,C 180,E1 -3290.474,E2 -3290.474} C_VEL
LIN {X 0,Y 552.114,Z 476.527,A -85,B 0,C 180,E1 -3293.316,E2 -3293.316} C_VEL
LIN {X 0,Y 552.131,Z 476.526,A -85,B 0,C 180,E1 -3295.94,E2 -3295.94} C_VEL
LIN {X 0,Y 552.147,Z 476.553,A -85,B 0,C 180,E1 -3297.594,E2 -3297.594} C_VEL
LIN {X 0,Y 552.702,Z 480.847,A -85,B 0,C 180,E1 -3299.004,E2 -3299.004} C_VEL
LIN {X 0,Y 552.578,Z 488.373,A -85,B 0,C 180,E1 -3301.352,E2 -3301.352} C_VEL
LIN {X 0,Y 552.456,Z 497.064,A -85,B 0,C 180,E1 -3303.968,E2 -3303.968} C_VEL
LIN {X 0,Y 552.286,Z 506.671,A -85,B 0,C 180,E1 -3306.767,E2 -3306.767} C_VEL
LIN {X 0,Y 552.188,Z 516.24,A -85,B 0,C 180,E1 -3309.513,E2 -3309.513} C_VEL
LIN {X 0,Y 552.107,Z 525.8,A -85,B 0,C 180,E1 -3312.212,E2 -3312.212} C_VEL
LIN {X 0,Y 551.976,Z 537.184,A -85,B 0,C 180,E1 -3315.39,E2 -3315.39} C_VEL
LIN {X 0,Y 551.901,Z 549.114,A -85,B 0,C 180,E1 -3318.675,E2 -3318.675} C_VEL
LIN {X 0,Y 551.851,Z 552.978,A -85,B 0,C 180,E1 -3319.73,E2 -3319.73} C_VEL
LIN {X 0,Y 552.51,Z 560.426,A -85,B 0,C 180,E1 -3319.927,E2 -3319.927} C_VEL
LIN {X 0,Y 552.459,Z 568.898,A -85,B 0,C 180,E1 -3320.204,E2 -3320.204} C_VEL
LIN {X 0,Y 552.394,Z 577.402,A -85,B 0,C 180,E1 -3320.573,E2 -3320.573} C_VEL
LIN {X 0,Y 552.279,Z 585.734,A -85,B 0,C 180,E1 -3321.032,E2 -3321.032} C_VEL
LIN {X 0,Y 552.188,Z 593.772,A -85,B 0,C 180,E1 -3321.584,E2 -3321.584} C_VEL
LIN {X 0,Y 552.066,Z 601.422,A -85,B 0,C 180,E1 -3322.227,E2 -3322.227} C_VEL
LIN {X 0,Y 551.987,Z 609.761,A -85,B 0,C 180,E1 -3323.09,E2 -3323.09} C_VEL
LIN {X 0,Y 551.944,Z 616.535,A -85,B 0,C 180,E1 -3323.986,E2 -3323.986} C_VEL
LIN {X 0,Y 551.747,Z 621.99,A -85,B 0,C 180,E1 -3324.885,E2 -3324.885} C_VEL
LIN {X 0,Y 551.779,Z 627.15,A -85,B 0,C 180,E1 -3325.983,E2 -3325.983} C_VEL
LIN {X 0,Y 551.731,Z 630.937,A -85,B 0,C 180,E1 -3327.08,E2 -3327.08} C_VEL
LIN {X 0,Y 551.657,Z 632.683,A -85,B 0,C 180,E1 -3327.81,E2 -3327.81} C_VEL
LIN {X 0,Y 551.644,Z 633.933,A -85,B 0,C 180,E1 -3328.54,E2 -3328.54} C_VEL
LIN {X 0,Y 551.639,Z 634.709,A -85,B 0,C 180,E1 -3329.27,E2 -3329.27} C_VEL
LIN {X 0,Y 551.638,Z 635,A -85,B 0,C 180,E1 -3330,E2 -3330} C_VEL
LIN {X 0,Y 551.639,Z 634.708,A -85,B 0,C 180,E1 -3330.73,E2 -3330.73} C_VEL
LIN {X 0,Y 551.644,Z 633.932,A -85,B 0,C 180,E1 -3331.46,E2 -3331.46} C_VEL
LIN {X 0,Y 551.657,Z 632.681,A -85,B 0,C 180,E1 -3332.191,E2 -3332.191} C_VEL
LIN {X 0,Y 551.768,Z 629.786,A -85,B 0,C 180,E1 -3333.286,E2 -3333.286} C_VEL
LIN {X 0,Y 551.773,Z 627.147,A -85,B 0,C 180,E1 -3334.017,E2 -3334.017} C_VEL
LIN {X 0,Y 551.747,Z 621.984,A -85,B 0,C 180,E1 -3335.116,E2 -3335.116} C_VEL
LIN {X 0,Y 551.957,Z 615.398,A -85,B 0,C 180,E1 -3336.184,E2 -3336.184} C_VEL
LIN {X 0,Y 551.994,Z 607.741,A -85,B 0,C 180,E1 -3337.131,E2 -3337.131} C_VEL
LIN {X 0,Y 552.076,Z 600.399,A -85,B 0,C 180,E1 -3337.866,E2 -3337.866} C_VEL
LIN {X 0,Y 552.229,Z 592.536,A -85,B 0,C 180,E1 -3338.508,E2 -3338.508} C_VEL
LIN {X 0,Y 552.306,Z 582.721,A -85,B 0,C 180,E1 -3339.153,E2 -3339.153} C_VEL
LIN {X 0,Y 552.458,Z 571.296,A -85,B 0,C 180,E1 -3339.704,E2 -3339.704} C_VEL
LIN {X 0,Y 552.544,Z 561.232,A -85,B 0,C 180,E1 -3340.05,E2 -3340.05} C_VEL
LIN {X 0,Y 551.833,Z 553.301,A -85,B 0,C 180,E1 -3340.271,E2 -3340.271} C_VEL
LIN {X 0,Y 551.859,Z 544.36,A -85,B 0,C 180,E1 -3342.878,E2 -3342.878} C_VEL
LIN {X 0,Y 551.965,Z 535.418,A -85,B 0,C 180,E1 -3345.509,E2 -3345.509} C_VEL
LIN {X 0,Y 552.073,Z 525.2,A -85,B 0,C 180,E1 -3348.558,E2 -3348.558} C_VEL
LIN {X 0,Y 552.123,Z 516.064,A -85,B 0,C 180,E1 -3351.271,E2 -3351.271} C_VEL
LIN {X 0,Y 552.219,Z 506.812,A -85,B 0,C 180,E1 -3354.033,E2 -3354.033} C_VEL
LIN {X 0,Y 552.379,Z 497.06,A -85,B 0,C 180,E1 -3357.049,E2 -3357.049} C_VEL
LIN {X 0,Y 552.49,Z 488.804,A -85,B 0,C 180,E1 -3359.743,E2 -3359.743} C_VEL
LIN {X 0,Y 552.727,Z 481.604,A -85,B 0,C 180,E1 -3362.279,E2 -3362.279} C_VEL
LIN {X 0,Y 552.292,Z 477.115,A -85,B 0,C 180,E1 -3364.05,E2 -3364.05} C_VEL
LIN {X 0,Y 552.164,Z 476.521,A -85,B 0,C 180,E1 -3364.372,E2 -3364.372} C_VEL
LIN {X 0,Y 552.096,Z 476.527,A -85,B 0,C 180,E1 -3367.664,E2 -3367.664} C_VEL
LIN {X 0,Y 552.122,Z 476.526,A -85,B 0,C 180,E1 -3370.48,E2 -3370.48} C_VEL
LIN {X 0,Y 552.122,Z 476.527,A -85,B 0,C 180,E1 -3373.485,E2 -3373.485} C_VEL
LIN {X 0,Y 552.123,Z 476.527,A -85,B 0,C 180,E1 -3376.578,E2 -3376.578} C_VEL
LIN {X 0,Y 552.113,Z 476.526,A -85,B 0,C 180,E1 -3379.519,E2 -3379.519} C_VEL
LIN {X 0,Y 552.096,Z 476.526,A -85,B 0,C 180,E1 -3382.336,E2 -3382.336} C_VEL
LIN {X 0,Y 552.086,Z 476.528,A -85,B 0,C 180,E1 -3385.051,E2 -3385.051} C_VEL
LIN {X 0,Y 552.074,Z 476.533,A -85,B 0,C 180,E1 -3387.679,E2 -3387.679} C_VEL
LIN {X 0,Y 552.004,Z 476.831,A -85,B 0,C 180,E1 -3388.543,E2 -3388.543} C_VEL
LIN {X 0,Y 551.921,Z 480.653,A -85,B 0,C 180,E1 -3391.478,E2 -3391.478} C_VEL
LIN {X 0,Y 551.853,Z 484.446,A -85,B 0,C 180,E1 -3394.342,E2 -3394.342} C_VEL
LIN {X 0,Y 551.808,Z 487.608,A -85,B 0,C 180,E1 -3396.745,E2 -3396.745} C_VEL
LIN {X 0,Y 551.748,Z 490.814,A -85,B 0,C 180,E1 -3399.105,E2 -3399.105} C_VEL
LIN {X 0,Y 551.714,Z 493.96,A -85,B 0,C 180,E1 -3401.43,E2 -3401.43} C_VEL
LIN {X 0,Y 551.718,Z 497.339,A -85,B 0,C 180,E1 -3403.725,E2 -3403.725} C_VEL
LIN {X 0,Y 551.716,Z 500.785,A -85,B 0,C 180,E1 -3405.994,E2 -3405.994} C_VEL
LIN {X 0,Y 551.72,Z 505.381,A -85,B 0,C 180,E1 -3408.985,E2 -3408.985} C_VEL
LIN {X 0,Y 551.706,Z 506.709,A -85,B 0,C 180,E1 -3409.843,E2 -3409.843} C_VEL
LIN {X 0,Y 552.526,Z 515.264,A -85,B 0,C 180,E1 -3410.112,E2 -3410.112} C_VEL
LIN {X 0,Y 552.411,Z 526.484,A -85,B 0,C 180,E1 -3410.572,E2 -3410.572} C_VEL
LIN {X 0,Y 552.269,Z 534.996,A -85,B 0,C 180,E1 -3411.032,E2 -3411.032} C_VEL
LIN {X 0,Y 552.172,Z 543.17,A -85,B 0,C 180,E1 -3411.583,E2 -3411.583} C_VEL
LIN {X 0,Y 552.071,Z 550.925,A -85,B 0,C 180,E1 -3412.226,E2 -3412.226} C_VEL
LIN {X 0,Y 551.97,Z 559.029,A -85,B 0,C 180,E1 -3413.053,E2 -3413.053} C_VEL
LIN {X 0,Y 551.931,Z 566.229,A -85,B 0,C 180,E1 -3413.983,E2 -3413.983} C_VEL
LIN {X 0,Y 551.747,Z 571.751,A -85,B 0,C 180,E1 -3414.885,E2 -3414.885} C_VEL
LIN {X 0,Y 551.81,Z 575.445,A -85,B 0,C 180,E1 -3415.617,E2 -3415.617} C_VEL
LIN {X 0,Y 551.769,Z 579.646,A -85,B 0,C 180,E1 -3416.714,E2 -3416.714} C_VEL
LIN {X 0,Y 551.655,Z 582.583,A -85,B 0,C 180,E1 -3417.81,E2 -3417.81} C_VEL
LIN {X 0,Y 551.645,Z 583.873,A -85,B 0,C 180,E1 -3418.54,E2 -3418.54} C_VEL
LIN {X 0,Y 551.638,Z 584.688,A -85,B 0,C 180,E1 -3419.27,E2 -3419.27} C_VEL
LIN {X 0,Y 551.637,Z 584.996,A -85,B 0,C 180,E1 -3420,E2 -3420} C_VEL
LIN {X 0,Y 551.64,Z 584.728,A -85,B 0,C 180,E1 -3420.73,E2 -3420.73} C_VEL
LIN {X 0,Y 551.644,Z 583.992,A -85,B 0,C 180,E1 -3421.46,E2 -3421.46} C_VEL
LIN {X 0,Y 551.656,Z 582.781,A -85,B 0,C 180,E1 -3422.19,E2 -3422.19} C_VEL
LIN {X 0,Y 551.756,Z 579.929,A -85,B 0,C 180,E1 -3423.286,E2 -3423.286} C_VEL
LIN {X 0,Y 551.774,Z 577.335,A -85,B 0,C 180,E1 -3424.017,E2 -3424.017} C_VEL
LIN {X 0,Y 551.738,Z 572.223,A -85,B 0,C 180,E1 -3425.116,E2 -3425.116} C_VEL
LIN {X 0,Y 551.928,Z 566.84,A -85,B 0,C 180,E1 -3426.012,E2 -3426.012} C_VEL
LIN {X 0,Y 551.945,Z 560.135,A -85,B 0,C 180,E1 -3426.911,E2 -3426.911} C_VEL
LIN {X 0,Y 552.044,Z 551.913,A -85,B 0,C 180,E1 -3427.774,E2 -3427.774} C_VEL
LIN {X 0,Y 552.157,Z 544.365,A -85,B 0,C 180,E1 -3428.417,E2 -3428.417} C_VEL
LIN {X 0,Y 552.272,Z 536.457,A -85,B 0,C 180,E1 -3428.968,E2 -3428.968} C_VEL
LIN {X 0,Y 552.376,Z 528.305,A -85,B 0,C 180,E1 -3429.428,E2 -3429.428} C_VEL
LIN {X 0,Y 552.455,Z 520.063,A -85,B 0,C 180,E1 -3429.797,E2 -3429.797} C_VEL
LIN {X 0,Y 552.345,Z 511.61,A -85,B 0,C 180,E1 -3430.088,E2 -3430.088} C_VEL
LIN {X 0,Y 551.712,Z 506.517,A -85,B 0,C 180,E1 -3430.25,E2 -3430.25} C_VEL
LIN {X 0,Y 551.705,Z 502.811,A -85,B 0,C 180,E1 -3432.507,E2 -3432.507} C_VEL
LIN {X 0,Y 551.736,Z 497.92,A -85,B 0,C 180,E1 -3435.515,E2 -3435.515} C_VEL
LIN {X 0,Y 551.706,Z 494.252,A -85,B 0,C 180,E1 -3437.802,E2 -3437.802} C_VEL
LIN {X 0,Y 551.754,Z 490.63,A -85,B 0,C 180,E1 -3440.116,E2 -3440.116} C_VEL
LIN {X 0,Y 551.776,Z 487.189,A -85,B 0,C 180,E1 -3442.465,E2 -3442.465} C_VEL
LIN {X 0,Y 551.846,Z 482.958,A -85,B 0,C 180,E1 -3445.281,E2 -3445.281} C_VEL
LIN {X 0,Y 551.913,Z 479.924,A -85,B 0,C 180,E1 -3447.285,E2 -3447.285} C_VEL
LIN {X 0,Y 551.955,Z 486.877,A -85,B 0,C 180,E1 -3450.021,E2 -3450.021} C_VEL
LIN {X 0,Y 551.947,Z 487.104,A -85,B 0,C 180,E1 -3450.113,E2 -3450.113} C_VEL
LIN {X 0,Y 551.255,Z 488.621,A -85,B 0,C 180,E1 -3450.702,E2 -3450.702} C_VEL
LIN {X 0,Y 548.403,Z 491.155,A -85,B 0,C 180,E1 -3451.655,E2 -3451.655} C_VEL
LIN {X 0,Y 546.005,Z 493.176,A -85,B 0,C 180,E1 -3452.423,E2 -3452.423} C_VEL
LIN {X 0,Y 544.971,Z 494.661,A -85,B 0,C 180,E1 -3453.017,E2 -3453.017} C_VEL
LIN {X 0,Y 544.884,Z 495.143,A -85,B 0,C 180,E1 -3453.219,E2 -3453.219} C_VEL
LIN {X 0,Y 544.787,Z 502.725,A -85,B 0,C 180,E1 -3456.4,E2 -3456.4} C_VEL
LIN {X 0,Y 544.741,Z 509.696,A -85,B 0,C 180,E1 -3459.277,E2 -3459.277} C_VEL
LIN {X 0,Y 544.705,Z 516.487,A -85,B 0,C 180,E1 -3462.139,E2 -3462.139} C_VEL
LIN {X 0,Y 544.689,Z 522.867,A -85,B 0,C 180,E1 -3464.793,E2 -3464.793} C_VEL
LIN {X 0,Y 544.667,Z 525,A -85,B 0,C 180,E1 -3465.674,E2 -3465.674} C_VEL
LIN {X 0,Y 545.549,Z 533.63,A -85,B 0,C 180,E1 -3465.936,E2 -3465.936} C_VEL
LIN {X 0,Y 545.41,Z 545.943,A -85,B 0,C 180,E1 -3466.418,E2 -3466.418} C_VEL
LIN {X 0,Y 545.259,Z 555.014,A -85,B 0,C 180,E1 -3466.911,E2 -3466.911} C_VEL
LIN {X 0,Y 545.146,Z 562.758,A -85,B 0,C 180,E1 -3467.436,E2 -3467.436} C_VEL
LIN {X 0,Y 544.988,Z 571.564,A -85,B 0,C 180,E1 -3468.181,E2 -3468.181} C_VEL
LIN {X 0,Y 544.873,Z 578.183,A -85,B 0,C 180,E1 -3468.866,E2 -3468.866} C_VEL
LIN {X 0,Y 544.828,Z 583.799,A -85,B 0,C 180,E1 -3469.559,E2 -3469.559} C_VEL
LIN {X 0,Y 544.733,Z 590.203,A -85,B 0,C 180,E1 -3470.541,E2 -3470.541} C_VEL
LIN {X 0,Y 544.678,Z 595.116,A -85,B 0,C 180,E1 -3471.495,E2 -3471.495} C_VEL
LIN {X 0,Y 544.675,Z 598.393,A -85,B 0,C 180,E1 -3472.293,E2 -3472.293} C_VEL
LIN {X 0,Y 544.609,Z 601.105,A -85,B 0,C 180,E1 -3473.139,E2 -3473.139} C_VEL
LIN {X 0,Y 544.565,Z 603.834,A -85,B 0,C 180,E1 -3474.496,E2 -3474.496} C_VEL
LIN {X 0,Y 544.574,Z 604.871,A -85,B 0,C 180,E1 -3475.685,E2 -3475.685} C_VEL
LIN {X 0,Y 544.566,Z 604.568,A -85,B 0,C 180,E1 -3477.021,E2 -3477.021} C_VEL
LIN {X 0,Y 544.59,Z 603.157,A -85,B 0,C 180,E1 -3478.054,E2 -3478.054} C_VEL
LIN {X 0,Y 544.628,Z 601.174,A -85,B 0,C 180,E1 -3478.924,E2 -3478.924} C_VEL
LIN {X 0,Y 544.659,Z 596.696,A -85,B 0,C 180,E1 -3480.236,E2 -3480.236} C_VEL
LIN {X 0,Y 544.716,Z 591.458,A -85,B 0,C 180,E1 -3481.324,E2 -3481.324} C_VEL
LIN {X 0,Y 544.787,Z 586.644,A -85,B 0,C 180,E1 -3482.118,E2 -3482.118} C_VEL
LIN {X 0,Y 544.858,Z 579.916,A -85,B 0,C 180,E1 -3483.017,E2 -3483.017} C_VEL
LIN {X 0,Y 544.973,Z 572.789,A -85,B 0,C 180,E1 -3483.788,E2 -3483.788} C_VEL
LIN {X 0,Y 545.109,Z 564.837,A -85,B 0,C 180,E1 -3484.488,E2 -3484.488} C_VEL
LIN {X 0,Y 545.253,Z 555.743,A -85,B 0,C 180,E1 -3485.132,E2 -3485.132} C_VEL
LIN {X 0,Y 545.427,Z 544.313,A -85,B 0,C 180,E1 -3485.75,E2 -3485.75} C_VEL
LIN {X 0,Y 545.541,Z 533.492,A -85,B 0,C 180,E1 -3486.158,E2 -3486.158} C_VEL
LIN {X 0,Y 544.642,Z 525.246,A -85,B 0,C 180,E1 -3486.42,E2 -3486.42} C_VEL
LIN {X 0,Y 544.647,Z 519.806,A -85,B 0,C 180,E1 -3488.819,E2 -3488.819} C_VEL
LIN {X 0,Y 544.703,Z 514.496,A -85,B 0,C 180,E1 -3491.182,E2 -3491.182} C_VEL
LIN {X 0,Y 544.748,Z 509.324,A -85,B 0,C 180,E1 -3493.511,E2 -3493.511} C_VEL
LIN {X 0,Y 544.789,Z 504.135,A -85,B 0,C 180,E1 -3495.811,E2 -3495.811} C_VEL
LIN {X 0,Y 544.906,Z 497.434,A -85,B 0,C 180,E1 -3498.845,E2 -3498.845} C_VEL
LIN {X 0,Y 544.854,Z 490.686,A -85,B 0,C 180,E1 -3501.843,E2 -3501.843} C_VEL
LIN {X 0,Y 544.942,Z 483.914,A -85,B 0,C 180,E1 -3504.82,E2 -3504.82} C_VEL
LIN {X 0,Y 544.914,Z 477.425,A -85,B 0,C 180,E1 -3507.69,E2 -3507.69} C_VEL
LIN {X 0,Y 545.206,Z 477.385,A -85,B 0,C 180,E1 -3510,E2 -3510} C_VEL
LIN {X 0,Y 545.172,Z 477.391,A -85,B 0,C 180,E1 -3512.955,E2 -3512.955} C_VEL
LIN {X 0,Y 545.178,Z 477.389,A -85,B 0,C 180,E1 -3515.919,E2 -3515.919} C_VEL
LIN {X 0,Y 545.113,Z 477.398,A -85,B 0,C 180,E1 -3518.9,E2 -3518.9} C_VEL
LIN {X 0,Y 545.137,Z 477.394,A -85,B 0,C 180,E1 -3521.904,E2 -3521.904} C_VEL
LIN {X 0,Y 545.087,Z 477.401,A -85,B 0,C 180,E1 -3524.943,E2 -3524.943} C_VEL
LIN {X 0,Y 545.083,Z 477.402,A -85,B 0,C 180,E1 -3528.025,E2 -3528.025} C_VEL
LIN {X 0,Y 545.097,Z 477.4,A -85,B 0,C 180,E1 -3530.372,E2 -3530.372} C_VEL
LIN {X 0,Y 545.093,Z 477.399,A -85,B 0,C 180,E1 -3533.558,E2 -3533.558} C_VEL
LIN {X 0,Y 545.09,Z 477.4,A -85,B 0,C 180,E1 -3536,E2 -3536} C_VEL
LIN {X 0,Y 545.092,Z 477.402,A -85,B 0,C 180,E1 -3538.748,E2 -3538.748} C_VEL
LIN {X 0,Y 545.079,Z 477.402,A -85,B 0,C 180,E1 -3541.682,E2 -3541.682} C_VEL
LIN {X 0,Y 545.082,Z 477.402,A -85,B 0,C 180,E1 -3544.563,E2 -3544.563} C_VEL
LIN {X 0,Y 545.04,Z 477.408,A -85,B 0,C 180,E1 -3547.303,E2 -3547.303} C_VEL
LIN {X 0,Y 545.071,Z 477.402,A -85,B 0,C 180,E1 -3550.142,E2 -3550.142} C_VEL
LIN {X 0,Y 545.085,Z 477.402,A -85,B 0,C 180,E1 -3553.105,E2 -3553.105} C_VEL
LIN {X 0,Y 545.064,Z 477.404,A -85,B 0,C 180,E1 -3556.224,E2 -3556.224} C_VEL
LIN {X 0,Y 545.104,Z 477.4,A -85,B 0,C 180,E1 -3558.887,E2 -3558.887} C_VEL
LIN {X 0,Y 545.053,Z 477.405,A -85,B 0,C 180,E1 -3561.763,E2 -3561.763} C_VEL
LIN {X 0,Y 545.035,Z 477.407,A -85,B 0,C 180,E1 -3564.531,E2 -3564.531} C_VEL
LIN {X 0,Y 545.081,Z 477.403,A -85,B 0,C 180,E1 -3567.212,E2 -3567.212} C_VEL
LIN {X 0,Y 545.065,Z 477.405,A -85,B 0,C 180,E1 -3569.81,E2 -3569.81} C_VEL
LIN {X 0,Y 545.095,Z 477.399,A -85,B 0,C 180,E1 -3572.344,E2 -3572.344} C_VEL
LIN {X 0,Y 545.117,Z 477.395,A -85,B 0,C 180,E1 -3574.82,E2 -3574.82} C_VEL
LIN {X 0,Y 545.043,Z 477.405,A -85,B 0,C 180,E1 -3577.242,E2 -3577.242} C_VEL
LIN {X 0,Y 545.12,Z 477.397,A -85,B 0,C 180,E1 -3580.415,E2 -3580.415} C_VEL
LIN {X 0,Y 545.073,Z 477.403,A -85,B 0,C 180,E1 -3583.521,E2 -3583.521} C_VEL
LIN {X 0,Y 545.094,Z 477.4,A -85,B 0,C 180,E1 -3585.82,E2 -3585.82} C_VEL
LIN {X 0,Y 545.116,Z 477.397,A -85,B 0,C 180,E1 -3588.849,E2 -3588.849} C_VEL
LIN {X 0,Y 545.129,Z 477.396,A -85,B 0,C 180,E1 -3591.847,E2 -3591.847} C_VEL
LIN {X 0,Y 545.203,Z 477.385,A -85,B 0,C 180,E1 -3594.823,E2 -3594.823} C_VEL
LIN {X 0,Y 545.196,Z 477.388,A -85,B 0,C 180,E1 -3597.784,E2 -3597.784} C_VEL
LIN {X 0,Y 545.212,Z 477.384,A -85,B 0,C 180,E1 -3600.739,E2 -3600.739} C_VEL
LIN {X 0,Y 545.174,Z 477.39,A -85,B 0,C 180,E1 -3602.956,E2 -3602.956} C_VEL
LIN {X 0,Y 545.172,Z 477.391,A -85,B 0,C 180,E1 -3605.919,E2 -3605.919} C_VEL
LIN {X 0,Y 545.12,Z 477.397,A -85,B 0,C 180,E1 -3608.9,E2 -3608.9} C_VEL
LIN {X 0,Y 545.133,Z 477.396,A -85,B 0,C 180,E1 -3611.904,E2 -3611.904} C_VEL
LIN {X 0,Y 545.084,Z 477.401,A -85,B 0,C 180,E1 -3614.944,E2 -3614.944} C_VEL
LIN {X 0,Y 545.082,Z 477.404,A -85,B 0,C 180,E1 -3618.026,E2 -3618.026} C_VEL
LIN {X 0,Y 545.093,Z 477.402,A -85,B 0,C 180,E1 -3620.372,E2 -3620.372} C_VEL
LIN {X 0,Y 545.09,Z 477.4,A -85,B 0,C 180,E1 -3623.559,E2 -3623.559} C_VEL
LIN {X 0,Y 545.078,Z 477.402,A -85,B 0,C 180,E1 -3626.001,E2 -3626.001} C_VEL
LIN {X 0,Y 545.09,Z 477.402,A -85,B 0,C 180,E1 -3628.749,E2 -3628.749} C_VEL
LIN {X 0,Y 545.076,Z 477.402,A -85,B 0,C 180,E1 -3631.683,E2 -3631.683} C_VEL
LIN {X 0,Y 545.08,Z 477.403,A -85,B 0,C 180,E1 -3634.563,E2 -3634.563} C_VEL
LIN {X 0,Y 545.038,Z 477.407,A -85,B 0,C 180,E1 -3637.304,E2 -3637.304} C_VEL
LIN {X 0,Y 545.067,Z 477.403,A -85,B 0,C 180,E1 -3640.142,E2 -3640.142} C_VEL
LIN {X 0,Y 545.087,Z 477.402,A -85,B 0,C 180,E1 -3643.106,E2 -3643.106} C_VEL
LIN {X 0,Y 545.055,Z 477.406,A -85,B 0,C 180,E1 -3646.226,E2 -3646.226} C_VEL
LIN {X 0,Y 545.1,Z 477.401,A -85,B 0,C 180,E1 -3648.888,E2 -3648.888} C_VEL
LIN {X 0,Y 545.053,Z 477.405,A -85,B 0,C 180,E1 -3651.763,E2 -3651.763} C_VEL
LIN {X 0,Y 545.065,Z 477.405,A -85,B 0,C 180,E1 -3654.534,E2 -3654.534} C_VEL
LIN {X 0,Y 545.125,Z 477.484,A -85,B 0,C 180,E1 -3657.435,E2 -3657.435} C_VEL
LIN {X 0,Y 545.747,Z 482.176,A -85,B 0,C 180,E1 -3658.996,E2 -3658.996} C_VEL
LIN {X 0,Y 545.572,Z 490.219,A -85,B 0,C 180,E1 -3661.535,E2 -3661.535} C_VEL
LIN {X 0,Y 545.451,Z 498.371,A -85,B 0,C 180,E1 -3664.019,E2 -3664.019} C_VEL
LIN {X 0,Y 545.243,Z 507.942,A -85,B 0,C 180,E1 -3666.851,E2 -3666.851} C_VEL
LIN {X 0,Y 545.124,Z 517.467,A -85,B 0,C 180,E1 -3669.629,E2 -3669.629} C_VEL
LIN {X 0,Y 545.008,Z 528.004,A -85,B 0,C 180,E1 -3672.601,E2 -3672.601} C_VEL
LIN {X 0,Y 544.904,Z 537.599,A -85,B 0,C 180,E1 -3675.313,E2 -3675.313} C_VEL
LIN {X 0,Y 544.82,Z 549.489,A -85,B 0,C 180,E1 -3678.63,E2 -3678.63} C_VEL
LIN {X 0,Y 544.773,Z 552.978,A -85,B 0,C 180,E1 -3679.595,E2 -3679.595} C_VEL
LIN {X 0,Y 545.536,Z 561.256,A -85,B 0,C 180,E1 -3679.821,E2 -3679.821} C_VEL
LIN {X 0,Y 545.444,Z 571.314,A -85,B 0,C 180,E1 -3680.17,E2 -3680.17} C_VEL
LIN {X 0,Y 545.318,Z 582.731,A -85,B 0,C 180,E1 -3680.73,E2 -3680.73} C_VEL
LIN {X 0,Y 545.21,Z 591.312,A -85,B 0,C 180,E1 -3681.289,E2 -3681.289} C_VEL
LIN {X 0,Y 545.044,Z 599.38,A -85,B 0,C 180,E1 -3681.939,E2 -3681.939} C_VEL
LIN {X 0,Y 544.932,Z 606.041,A -85,B 0,C 180,E1 -3682.59,E2 -3682.59} C_VEL
LIN {X 0,Y 544.839,Z 612.361,A -85,B 0,C 180,E1 -3683.334,E2 -3683.334} C_VEL
LIN {X 0,Y 544.843,Z 617.613,A -85,B 0,C 180,E1 -3684.077,E2 -3684.077} C_VEL
LIN {X 0,Y 544.673,Z 621.991,A -85,B 0,C 180,E1 -3684.818,E2 -3684.818} C_VEL
LIN {X 0,Y 544.702,Z 627.15,A -85,B 0,C 180,E1 -3685.931,E2 -3685.931} C_VEL
LIN {X 0,Y 544.66,Z 630.937,A -85,B 0,C 180,E1 -3687.042,E2 -3687.042} C_VEL
LIN {X 0,Y 544.571,Z 632.683,A -85,B 0,C 180,E1 -3687.782,E2 -3687.782} C_VEL
LIN {X 0,Y 544.545,Z 633.932,A -85,B 0,C 180,E1 -3688.521,E2 -3688.521} C_VEL
LIN {X 0,Y 544.54,Z 634.708,A -85,B 0,C 180,E1 -3689.261,E2 -3689.261} C_VEL
LIN {X 0,Y 544.538,Z 635,A -85,B 0,C 180,E1 -3690,E2 -3690} C_VEL
LIN {X 0,Y 544.54,Z 634.708,A -85,B 0,C 180,E1 -3690.74,E2 -3690.74} C_VEL
LIN {X 0,Y 544.545,Z 633.931,A -85,B 0,C 180,E1 -3691.479,E2 -3691.479} C_VEL
LIN {X 0,Y 544.572,Z 632.681,A -85,B 0,C 180,E1 -3692.219,E2 -3692.219} C_VEL
LIN {X 0,Y 544.695,Z 629.786,A -85,B 0,C 180,E1 -3693.329,E2 -3693.329} C_VEL
LIN {X 0,Y 544.697,Z 627.147,A -85,B 0,C 180,E1 -3694.07,E2 -3694.07} C_VEL
LIN {X 0,Y 544.673,Z 621.984,A -85,B 0,C 180,E1 -3695.183,E2 -3695.183} C_VEL
LIN {X 0,Y 544.88,Z 615.956,A -85,B 0,C 180,E1 -3696.183,E2 -3696.183} C_VEL
LIN {X 0,Y 544.922,Z 607.74,A -85,B 0,C 180,E1 -3697.224,E2 -3697.224} C_VEL
LIN {X 0,Y 545.036,Z 600.397,A -85,B 0,C 180,E1 -3697.968,E2 -3697.968} C_VEL
LIN {X 0,Y 545.201,Z 592.533,A -85,B 0,C 180,E1 -3698.619,E2 -3698.619} C_VEL
LIN {X 0,Y 545.268,Z 584.22,A -85,B 0,C 180,E1 -3699.178,E2 -3699.178} C_VEL
LIN {X 0,Y 545.433,Z 573.603,A -85,B 0,C 180,E1 -3699.737,E2 -3699.737} C_VEL
LIN {X 0,Y 545.547,Z 562.063,A -85,B 0,C 180,E1 -3700.156,E2 -3700.156} C_VEL
LIN {X 0,Y 544.737,Z 553.301,A -85,B 0,C 180,E1 -3700.406,E2 -3700.406} C_VEL
LIN {X 0,Y 544.802,Z 544.36,A -85,B 0,C 180,E1 -3703.047,E2 -3703.047} C_VEL
LIN {X 0,Y 544.894,Z 535.418,A -85,B 0,C 180,E1 -3705.716,E2 -3705.716} C_VEL
LIN {X 0,Y 545.012,Z 526.362,A -85,B 0,C 180,E1 -3708.417,E2 -3708.417} C_VEL
LIN {X 0,Y 545.054,Z 517.079,A -85,B 0,C 180,E1 -3711.164,E2 -3711.164} C_VEL
LIN {X 0,Y 545.162,Z 507.688,A -85,B 0,C 180,E1 -3714.02,E2 -3714.02} C_VEL
LIN {X 0,Y 545.309,Z 498.794,A -85,B 0,C 180,E1 -3716.814,E2 -3716.814} C_VEL
LIN {X 0,Y 545.454,Z 491.209,A -85,B 0,C 180,E1 -3719.316,E2 -3719.316} C_VEL
LIN {X 0,Y 545.745,Z 482.853,A -85,B 0,C 180,E1 -3722.306,E2 -3722.306} C_VEL
LIN {X 0,Y 545.487,Z 479.507,A -85,B 0,C 180,E1 -3723.643,E2 -3723.643} C_VEL
LIN {X 0,Y 545.098,Z 477.401,A -85,B 0,C 180,E1 -3724.562,E2 -3724.562} C_VEL
LIN {X 0,Y 545.041,Z 477.408,A -85,B 0,C 180,E1 -3727.304,E2 -3727.304} C_VEL
LIN {X 0,Y 545.074,Z 477.405,A -85,B 0,C 180,E1 -3730.142,E2 -3730.142} C_VEL
LIN {X 0,Y 545.081,Z 477.402,A -85,B 0,C 180,E1 -3733.107,E2 -3733.107} C_VEL
LIN {X 0,Y 545.068,Z 477.403,A -85,B 0,C 180,E1 -3736.225,E2 -3736.225} C_VEL
LIN {X 0,Y 545.09,Z 477.398,A -85,B 0,C 180,E1 -3738.886,E2 -3738.886} C_VEL
LIN {X 0,Y 545.055,Z 477.405,A -85,B 0,C 180,E1 -3741.763,E2 -3741.763} C_VEL
LIN {X 0,Y 545.039,Z 477.409,A -85,B 0,C 180,E1 -3744.532,E2 -3744.532} C_VEL
LIN {X 0,Y 545.059,Z 477.404,A -85,B 0,C 180,E1 -3747.211,E2 -3747.211} C_VEL
LIN {X 0,Y 544.949,Z 477.448,A -85,B 0,C 180,E1 -3748.341,E2 -3748.341} C_VEL
LIN {X 0,Y 544.875,Z 481.22,A -85,B 0,C 180,E1 -3751.294,E2 -3751.294} C_VEL
LIN {X 0,Y 544.782,Z 484.717,A -85,B 0,C 180,E1 -3753.984,E2 -3753.984} C_VEL
LIN {X 0,Y 544.748,Z 487.925,A -85,B 0,C 180,E1 -3756.425,E2 -3756.425} C_VEL
LIN {X 0,Y 544.698,Z 492.201,A -85,B 0,C 180,E1 -3759.612,E2 -3759.612} C_VEL
LIN {X 0,Y 544.663,Z 496.378,A -85,B 0,C 180,E1 -3762.718,E2 -3762.718} C_VEL
LIN {X 0,Y 544.659,Z 500.191,A -85,B 0,C 180,E1 -3765.413,E2 -3765.413} C_VEL
LIN {X 0,Y 544.629,Z 505.382,A -85,B 0,C 180,E1 -3768.839,E2 -3768.839} C_VEL
LIN {X 0,Y 544.615,Z 506.71,A -85,B 0,C 180,E1 -3769.709,E2 -3769.709} C_VEL
LIN {X 0,Y 545.526,Z 515.279,A -85,B 0,C 180,E1 -3769.984,E2 -3769.984} C_VEL
LIN {X 0,Y 545.423,Z 524.622,A -85,B 0,C 180,E1 -3770.357,E2 -3770.357} C_VEL
LIN {X 0,Y 545.241,Z 535.004,A -85,B 0,C 180,E1 -3770.915,E2 -3770.915} C_VEL
LIN {X 0,Y 545.157,Z 543.175,A -85,B 0,C 180,E1 -3771.474,E2 -3771.474} C_VEL
LIN {X 0,Y 545.036,Z 550.929,A -85,B 0,C 180,E1 -3772.125,E2 -3772.125} C_VEL
LIN {X 0,Y 544.921,Z 559.034,A -85,B 0,C 180,E1 -3772.963,E2 -3772.963} C_VEL
LIN {X 0,Y 544.891,Z 565.635,A -85,B 0,C 180,E1 -3773.815,E2 -3773.815} C_VEL
LIN {X 0,Y 544.673,Z 571.754,A -85,B 0,C 180,E1 -3774.818,E2 -3774.818} C_VEL
LIN {X 0,Y 544.712,Z 575.448,A -85,B 0,C 180,E1 -3775.56,E2 -3775.56} C_VEL
LIN {X 0,Y 544.697,Z 579.647,A -85,B 0,C 180,E1 -3776.671,E2 -3776.671} C_VEL
LIN {X 0,Y 544.57,Z 582.583,A -85,B 0,C 180,E1 -3777.781,E2 -3777.781} C_VEL
LIN {X 0,Y 544.546,Z 583.872,A -85,B 0,C 180,E1 -3778.521,E2 -3778.521} C_VEL
LIN {X 0,Y 544.539,Z 584.688,A -85,B 0,C 180,E1 -3779.261,E2 -3779.261} C_VEL
LIN {X 0,Y 544.537,Z 584.996,A -85,B 0,C 180,E1 -3780,E2 -3780} C_VEL
LIN {X 0,Y 544.54,Z 584.727,A -85,B 0,C 180,E1 -3780.74,E2 -3780.74} C_VEL
LIN {X 0,Y 544.545,Z 583.99,A -85,B 0,C 180,E1 -3781.479,E2 -3781.479} C_VEL
LIN {X 0,Y 544.571,Z 582.78,A -85,B 0,C 180,E1 -3782.219,E2 -3782.219} C_VEL
LIN {X 0,Y 544.684,Z 579.927,A -85,B 0,C 180,E1 -3783.329,E2 -3783.329} C_VEL
LIN {X 0,Y 544.698,Z 577.333,A -85,B 0,C 180,E1 -3784.069,E2 -3784.069} C_VEL
LIN {X 0,Y 544.668,Z 572.22,A -85,B 0,C 180,E1 -3785.182,E2 -3785.182} C_VEL
LIN {X 0,Y 544.883,Z 566.268,A -85,B 0,C 180,E1 -3786.18,E2 -3786.18} C_VEL
LIN {X 0,Y 544.921,Z 558.152,A -85,B 0,C 180,E1 -3787.224,E2 -3787.224} C_VEL
LIN {X 0,Y 545.003,Z 550.887,A -85,B 0,C 180,E1 -3787.968,E2 -3787.968} C_VEL
LIN {X 0,Y 545.177,Z 543.126,A -85,B 0,C 180,E1 -3788.619,E2 -3788.619} C_VEL
LIN {X 0,Y 545.267,Z 534.945,A -85,B 0,C 180,E1 -3789.178,E2 -3789.178} C_VEL
LIN {X 0,Y 545.44,Z 524.544,A -85,B 0,C 180,E1 -3789.736,E2 -3789.736} C_VEL
LIN {X 0,Y 545.411,Z 512.835,A -85,B 0,C 180,E1 -3790.182,E2 -3790.182} C_VEL
LIN {X 0,Y 544.622,Z 506.516,A -85,B 0,C 180,E1 -3790.385,E2 -3790.385} C_VEL
LIN {X 0,Y 544.615,Z 501.587,A -85,B 0,C 180,E1 -3793.431,E2 -3793.431} C_VEL
LIN {X 0,Y 544.638,Z 497.919,A -85,B 0,C 180,E1 -3795.723,E2 -3795.723} C_VEL
LIN {X 0,Y 544.632,Z 494.331,A -85,B 0,C 180,E1 -3798.041,E2 -3798.041} C_VEL
LIN {X 0,Y 544.683,Z 490.862,A -85,B 0,C 180,E1 -3800.388,E2 -3800.388} C_VEL
LIN {X 0,Y 544.709,Z 487.382,A -85,B 0,C 180,E1 -3802.772,E2 -3802.772} C_VEL
LIN {X 0,Y 544.782,Z 483.308,A -85,B 0,C 180,E1 -3805.439,E2 -3805.439} C_VEL
LIN {X 0,Y 544.848,Z 480.634,A -85,B 0,C 180,E1 -3807.323,E2 -3807.323} C_VEL
LIN {X 0,Y 544.878,Z 486.772,A -85,B 0,C 180,E1 -3809.774,E2 -3809.774} C_VEL
LIN {X 0,Y 544.9,Z 493.125,A -85,B 0,C 180,E1 -3812.361,E2 -3812.361} C_VEL
LIN {X 0,Y 544.884,Z 495.143,A -85,B 0,C 180,E1 -3813.219,E2 -3813.219} C_VEL
LIN {X 0,Y 544.193,Z 496.614,A -85,B 0,C 180,E1 -3813.816,E2 -3813.816} C_VEL
LIN {X 0,Y 541.28,Z 499.141,A -85,B 0,C 180,E1 -3814.78,E2 -3814.78} C_VEL
LIN {X 0,Y 538.835,Z 501.18,A -85,B 0,C 180,E1 -3815.556,E2 -3815.556} C_VEL
LIN {X 0,Y 537.803,Z 502.694,A -85,B 0,C 180,E1 -3816.157,E2 -3816.157} C_VEL
LIN {X 0,Y 537.727,Z 503.188,A -85,B 0,C 180,E1 -3816.361,E2 -3816.361} C_VEL
LIN {X 0,Y 537.677,Z 510.881,A -85,B 0,C 180,E1 -3819.539,E2 -3819.539} C_VEL
LIN {X 0,Y 537.609,Z 517.353,A -85,B 0,C 180,E1 -3822.317,E2 -3822.317} C_VEL
LIN {X 0,Y 537.594,Z 523.943,A -85,B 0,C 180,E1 -3825.094,E2 -3825.094} C_VEL
LIN {X 0,Y 537.603,Z 524.995,A -85,B 0,C 180,E1 -3825.534,E2 -3825.534} C_VEL
LIN {X 0,Y 538.562,Z 533.805,A -85,B 0,C 180,E1 -3825.809,E2 -3825.809} C_VEL
LIN {X 0,Y 538.411,Z 545.697,A -85,B 0,C 180,E1 -3826.279,E2 -3826.279} C_VEL
LIN {X 0,Y 538.22,Z 555.838,A -85,B 0,C 180,E1 -3826.845,E2 -3826.845} C_VEL
LIN {X 0,Y 538.088,Z 564.556,A -85,B 0,C 180,E1 -3827.468,E2 -3827.468} C_VEL
LIN {X 0,Y 537.923,Z 572.121,A -85,B 0,C 180,E1 -3828.134,E2 -3828.134} C_VEL
LIN {X 0,Y 537.819,Z 578.664,A -85,B 0,C 180,E1 -3828.831,E2 -3828.831} C_VEL
LIN {X 0,Y 537.743,Z 584.066,A -85,B 0,C 180,E1 -3829.512,E2 -3829.512} C_VEL
LIN {X 0,Y 537.671,Z 590.161,A -85,B 0,C 180,E1 -3830.462,E2 -3830.462} C_VEL
LIN {X 0,Y 537.605,Z 595.074,A -85,B 0,C 180,E1 -3831.427,E2 -3831.427} C_VEL
LIN {X 0,Y 537.571,Z 597.856,A -85,B 0,C 180,E1 -3832.087,E2 -3832.087} C_VEL
LIN {X 0,Y 537.511,Z 600.905,A -85,B 0,C 180,E1 -3833.026,E2 -3833.026} C_VEL
LIN {X 0,Y 537.456,Z 603.41,A -85,B 0,C 180,E1 -3834.168,E2 -3834.168} C_VEL
LIN {X 0,Y 537.454,Z 604.367,A -85,B 0,C 180,E1 -3834.874,E2 -3834.874} C_VEL
LIN {X 0,Y 537.472,Z 604.917,A -85,B 0,C 180,E1 -3835.787,E2 -3835.787} C_VEL
LIN {X 0,Y 537.465,Z 604.686,A -85,B 0,C 180,E1 -3836.812,E2 -3836.812} C_VEL
LIN {X 0,Y 537.505,Z 602.914,A -85,B 0,C 180,E1 -3838.2,E2 -3838.2} C_VEL
LIN {X 0,Y 537.566,Z 600.043,A -85,B 0,C 180,E1 -3839.344,E2 -3839.344} C_VEL
LIN {X 0,Y 537.561,Z 597.033,A -85,B 0,C 180,E1 -3840.211,E2 -3840.211} C_VEL
LIN {X 0,Y 537.624,Z 591.731,A -85,B 0,C 180,E1 -3841.343,E2 -3841.343} C_VEL
LIN {X 0,Y 537.7,Z 587.036,A -85,B 0,C 180,E1 -3842.14,E2 -3842.14} C_VEL
LIN {X 0,Y 537.798,Z 580.873,A -85,B 0,C 180,E1 -3842.992,E2 -3842.992} C_VEL
LIN {X 0,Y 537.85,Z 575.458,A -85,B 0,C 180,E1 -3843.623,E2 -3843.623} C_VEL
LIN {X 0,Y 538.006,Z 568.035,A -85,B 0,C 180,E1 -3844.336,E2 -3844.336} C_VEL
LIN {X 0,Y 538.17,Z 559.667,A -85,B 0,C 180,E1 -3844.989,E2 -3844.989} C_VEL
LIN {X 0,Y 538.283,Z 551.413,A -85,B 0,C 180,E1 -3845.51,E2 -3845.51} C_VEL
LIN {X 0,Y 538.445,Z 542.59,A -85,B 0,C 180,E1 -3845.948,E2 -3845.948} C_VEL
LIN {X 0,Y 538.488,Z 532.85,A -85,B 0,C 180,E1 -3846.311,E2 -3846.311} C_VEL
LIN {X 0,Y 537.537,Z 525.268,A -85,B 0,C 180,E1 -3846.549,E2 -3846.549} C_VEL
LIN {X 0,Y 537.569,Z 519.052,A -85,B 0,C 180,E1 -3849.329,E2 -3849.329} C_VEL
LIN {X 0,Y 537.623,Z 513.819,A -85,B 0,C 180,E1 -3851.715,E2 -3851.715} C_VEL
LIN {X 0,Y 537.648,Z 508.595,A -85,B 0,C 180,E1 -3854.067,E2 -3854.067} C_VEL
LIN {X 0,Y 537.691,Z 503.352,A -85,B 0,C 180,E1 -3856.392,E2 -3856.392} C_VEL
LIN {X 0,Y 537.834,Z 498.33,A -85,B 0,C 180,E1 -3858.696,E2 -3858.696} C_VEL
LIN {X 0,Y 537.793,Z 491.56,A -85,B 0,C 180,E1 -3861.735,E2 -3861.735} C_VEL
LIN {X 0,Y 537.873,Z 484.743,A -85,B 0,C 180,E1 -3864.752,E2 -3864.752} C_VEL
LIN {X 0,Y 537.83,Z 478.307,A -85,B 0,C 180,E1 -3867.659,E2 -3867.659} C_VEL
LIN {X 0,Y 538.184,Z 478.262,A -85,B 0,C 180,E1 -3869.251,E2 -3869.251} C_VEL
LIN {X 0,Y 538.171,Z 478.262,A -85,B 0,C 180,E1 -3872.245,E2 -3872.245} C_VEL
LIN {X 0,Y 538.166,Z 478.264,A -85,B 0,C 180,E1 -3875.245,E2 -3875.245} C_VEL
LIN {X 0,Y 538.086,Z 478.272,A -85,B 0,C 180,E1 -3878.26,E2 -3878.26} C_VEL
LIN {X 0,Y 538.091,Z 478.272,A -85,B 0,C 180,E1 -3881.6,E2 -3881.6} C_VEL
LIN {X 0,Y 538.06,Z 478.276,A -85,B 0,C 180,E1 -3884.857,E2 -3884.857} C_VEL
LIN {X 0,Y 538.06,Z 478.275,A -85,B 0,C 180,E1 -3887.54,E2 -3887.54} C_VEL
LIN {X 0,Y 538.041,Z 478.28,A -85,B 0,C 180,E1 -3890.651,E2 -3890.651} C_VEL
LIN {X 0,Y 538.025,Z 478.28,A -85,B 0,C 180,E1 -3893.887,E2 -3893.887} C_VEL
LIN {X 0,Y 538.051,Z 478.279,A -85,B 0,C 180,E1 -3896.366,E2 -3896.366} C_VEL
LIN {X 0,Y 538.038,Z 478.28,A -85,B 0,C 180,E1 -3898.934,E2 -3898.934} C_VEL
LIN {X 0,Y 538.028,Z 478.28,A -85,B 0,C 180,E1 -3901.89,E2 -3901.89} C_VEL
LIN {X 0,Y 538.032,Z 478.281,A -85,B 0,C 180,E1 -3904.62,E2 -3904.62} C_VEL
LIN {X 0,Y 538.008,Z 478.284,A -85,B 0,C 180,E1 -3907.17,E2 -3907.17} C_VEL
LIN {X 0,Y 538.027,Z 478.281,A -85,B 0,C 180,E1 -3909.796,E2 -3909.796} C_VEL
LIN {X 0,Y 538.022,Z 478.281,A -85,B 0,C 180,E1 -3912.785,E2 -3912.785} C_VEL
LIN {X 0,Y 538.028,Z 478.28,A -85,B 0,C 180,E1 -3915.925,E2 -3915.925} C_VEL
LIN {X 0,Y 538.078,Z 478.274,A -85,B 0,C 180,E1 -3919.249,E2 -3919.249} C_VEL
LIN {X 0,Y 537.992,Z 478.285,A -85,B 0,C 180,E1 -3922.122,E2 -3922.122} C_VEL
LIN {X 0,Y 537.997,Z 478.285,A -85,B 0,C 180,E1 -3924.915,E2 -3924.915} C_VEL
LIN {X 0,Y 538.03,Z 478.28,A -85,B 0,C 180,E1 -3927.618,E2 -3927.618} C_VEL
LIN {X 0,Y 538.017,Z 478.281,A -85,B 0,C 180,E1 -3930.239,E2 -3930.239} C_VEL
LIN {X 0,Y 538.07,Z 478.275,A -85,B 0,C 180,E1 -3932.796,E2 -3932.796} C_VEL
LIN {X 0,Y 538.048,Z 478.277,A -85,B 0,C 180,E1 -3935.293,E2 -3935.293} C_VEL
LIN {X 0,Y 538.014,Z 478.283,A -85,B 0,C 180,E1 -3938.042,E2 -3938.042} C_VEL
LIN {X 0,Y 538.037,Z 478.277,A -85,B 0,C 180,E1 -3940.94,E2 -3940.94} C_VEL
LIN {X 0,Y 538.024,Z 478.28,A -85,B 0,C 180,E1 -3943.299,E2 -3943.299} C_VEL
LIN {X 0,Y 538.063,Z 478.275,A -85,B 0,C 180,E1 -3945.631,E2 -3945.631} C_VEL
LIN {X 0,Y 538.075,Z 478.275,A -85,B 0,C 180,E1 -3948.701,E2 -3948.701} C_VEL
LIN {X 0,Y 538.086,Z 478.273,A -85,B 0,C 180,E1 -3951.74,E2 -3951.74} C_VEL
LIN {X 0,Y 538.16,Z 478.263,A -85,B 0,C 180,E1 -3954.755,E2 -3954.755} C_VEL
LIN {X 0,Y 538.168,Z 478.264,A -85,B 0,C 180,E1 -3957.755,E2 -3957.755} C_VEL
LIN {X 0,Y 538.182,Z 478.26,A -85,B 0,C 180,E1 -3960.748,E2 -3960.748} C_VEL
LIN {X 0,Y 538.141,Z 478.266,A -85,B 0,C 180,E1 -3962.994,E2 -3962.994} C_VEL
LIN {X 0,Y 538.125,Z 478.269,A -85,B 0,C 180,E1 -3965.997,E2 -3965.997} C_VEL
LIN {X 0,Y 538.071,Z 478.274,A -85,B 0,C 180,E1 -3969.018,E2 -3969.018} C_VEL
LIN {X 0,Y 538.082,Z 478.276,A -85,B 0,C 180,E1 -3972.062,E2 -3972.062} C_VEL
LIN {X 0,Y 538.044,Z 478.277,A -85,B 0,C 180,E1 -3975.144,E2 -3975.144} C_VEL
LIN {X 0,Y 538.033,Z 478.279,A -85,B 0,C 180,E1 -3978.27,E2 -3978.27} C_VEL
LIN {X 0,Y 538.037,Z 478.279,A -85,B 0,C 180,E1 -3980.651,E2 -3980.651} C_VEL
LIN {X 0,Y 538.022,Z 478.283,A -85,B 0,C 180,E1 -3983.887,E2 -3983.887} C_VEL
LIN {X 0,Y 538.04,Z 478.28,A -85,B 0,C 180,E1 -3986.367,E2 -3986.367} C_VEL
LIN {X 0,Y 538.054,Z 478.277,A -85,B 0,C 180,E1 -3988.939,E2 -3988.939} C_VEL
LIN {X 0,Y 538.026,Z 478.281,A -85,B 0,C 180,E1 -3991.891,E2 -3991.891} C_VEL
LIN {X 0,Y 538.03,Z 478.281,A -85,B 0,C 180,E1 -3994.621,E2 -3994.621} C_VEL
LIN {X 0,Y 538.006,Z 478.284,A -85,B 0,C 180,E1 -3997.171,E2 -3997.171} C_VEL
LIN {X 0,Y 538.022,Z 478.28,A -85,B 0,C 180,E1 -3999.797,E2 -3999.797} C_VEL
LIN {X 0,Y 538.023,Z 478.282,A -85,B 0,C 180,E1 -4002.785,E2 -4002.785} C_VEL
LIN {X 0,Y 538.03,Z 478.281,A -85,B 0,C 180,E1 -4005.141,E2 -4005.141} C_VEL
LIN {X 0,Y 538.04,Z 478.278,A -85,B 0,C 180,E1 -4008.228,E2 -4008.228} C_VEL
LIN {X 0,Y 538.058,Z 478.275,A -85,B 0,C 180,E1 -4010.412,E2 -4010.412} C_VEL
LIN {X 0,Y 538.028,Z 478.28,A -85,B 0,C 180,E1 -4013.068,E2 -4013.068} C_VEL
LIN {X 0,Y 538.027,Z 478.283,A -85,B 0,C 180,E1 -4015.828,E2 -4015.828} C_VEL
LIN {X 0,Y 538.114,Z 478.471,A -85,B 0,C 180,E1 -4017.291,E2 -4017.291} C_VEL
LIN {X 0,Y 538.771,Z 483.479,A -85,B 0,C 180,E1 -4018.986,E2 -4018.986} C_VEL
LIN {X 0,Y 538.59,Z 491.522,A -85,B 0,C 180,E1 -4021.557,E2 -4021.557} C_VEL
LIN {X 0,Y 538.378,Z 500.987,A -85,B 0,C 180,E1 -4024.483,E2 -4024.483} C_VEL
LIN {X 0,Y 538.222,Z 510.533,A -85,B 0,C 180,E1 -4027.344,E2 -4027.344} C_VEL
LIN {X 0,Y 538.037,Z 520.052,A -85,B 0,C 180,E1 -4030.147,E2 -4030.147} C_VEL
LIN {X 0,Y 537.933,Z 529.724,A -85,B 0,C 180,E1 -4032.905,E2 -4032.905} C_VEL
LIN {X 0,Y 537.799,Z 540.748,A -85,B 0,C 180,E1 -4036.01,E2 -4036.01} C_VEL
LIN {X 0,Y 537.724,Z 551.619,A -85,B 0,C 180,E1 -4039.076,E2 -4039.076} C_VEL
LIN {X 0,Y 537.689,Z 552.978,A -85,B 0,C 180,E1 -4039.456,E2 -4039.456} C_VEL
LIN {X 0,Y 538.554,Z 562.087,A -85,B 0,C 180,E1 -4039.711,E2 -4039.711} C_VEL
LIN {X 0,Y 538.427,Z 573.616,A -85,B 0,C 180,E1 -4040.136,E2 -4040.136} C_VEL
LIN {X 0,Y 538.261,Z 584.229,A -85,B 0,C 180,E1 -4040.702,E2 -4040.702} C_VEL
LIN {X 0,Y 538.16,Z 592.538,A -85,B 0,C 180,E1 -4041.268,E2 -4041.268} C_VEL
LIN {X 0,Y 537.984,Z 600.398,A -85,B 0,C 180,E1 -4041.927,E2 -4041.927} C_VEL
LIN {X 0,Y 537.852,Z 607.743,A -85,B 0,C 180,E1 -4042.681,E2 -4042.681} C_VEL
LIN {X 0,Y 537.792,Z 614.664,A -85,B 0,C 180,E1 -4043.552,E2 -4043.552} C_VEL
LIN {X 0,Y 537.652,Z 621.033,A -85,B 0,C 180,E1 -4044.562,E2 -4044.562} C_VEL
LIN {X 0,Y 537.612,Z 625.634,A -85,B 0,C 180,E1 -4045.502,E2 -4045.502} C_VEL
LIN {X 0,Y 537.599,Z 628.622,A -85,B 0,C 180,E1 -4046.253,E2 -4046.253} C_VEL
LIN {X 0,Y 537.564,Z 630.938,A -85,B 0,C 180,E1 -4047.003,E2 -4047.003} C_VEL
LIN {X 0,Y 537.49,Z 632.682,A -85,B 0,C 180,E1 -4047.752,E2 -4047.752} C_VEL
LIN {X 0,Y 537.45,Z 633.931,A -85,B 0,C 180,E1 -4048.502,E2 -4048.502} C_VEL
LIN {X 0,Y 537.44,Z 634.707,A -85,B 0,C 180,E1 -4049.251,E2 -4049.251} C_VEL
LIN {X 0,Y 537.439,Z 635,A -85,B 0,C 180,E1 -4050,E2 -4050} C_VEL
LIN {X 0,Y 537.44,Z 634.707,A -85,B 0,C 180,E1 -4050.75,E2 -4050.75} C_VEL
LIN {X 0,Y 537.45,Z 633.93,A -85,B 0,C 180,E1 -4051.499,E2 -4051.499} C_VEL
LIN {X 0,Y 537.49,Z 632.68,A -85,B 0,C 180,E1 -4052.248,E2 -4052.248} C_VEL
LIN {X 0,Y 537.595,Z 629.785,A -85,B 0,C 180,E1 -4053.373,E2 -4053.373} C_VEL
LIN {X 0,Y 537.622,Z 627.147,A -85,B 0,C 180,E1 -4054.123,E2 -4054.123} C_VEL
LIN {X 0,Y 537.606,Z 621.984,A -85,B 0,C 180,E1 -4055.251,E2 -4055.251} C_VEL
LIN {X 0,Y 537.802,Z 616.198,A -85,B 0,C 180,E1 -4056.226,E2 -4056.226} C_VEL
LIN {X 0,Y 537.854,Z 609.432,A -85,B 0,C 180,E1 -4057.131,E2 -4057.131} C_VEL
LIN {X 0,Y 537.991,Z 601.416,A -85,B 0,C 180,E1 -4057.979,E2 -4057.979} C_VEL
LIN {X 0,Y 538.135,Z 593.761,A -85,B 0,C 180,E1 -4058.638,E2 -4058.638} C_VEL
LIN {X 0,Y 538.226,Z 585.718,A -85,B 0,C 180,E1 -4059.205,E2 -4059.205} C_VEL
LIN {X 0,Y 538.393,Z 577.384,A -85,B 0,C 180,E1 -4059.676,E2 -4059.676} C_VEL
LIN {X 0,Y 538.505,Z 568.878,A -85,B 0,C 180,E1 -4060.053,E2 -4060.053} C_VEL
LIN {X 0,Y 538.463,Z 559.984,A -85,B 0,C 180,E1 -4060.351,E2 -4060.351} C_VEL
LIN {X 0,Y 537.65,Z 553.301,A -85,B 0,C 180,E1 -4060.545,E2 -4060.545} C_VEL
LIN {X 0,Y 537.731,Z 544.36,A -85,B 0,C 180,E1 -4063.222,E2 -4063.222} C_VEL
LIN {X 0,Y 537.822,Z 535.307,A -85,B 0,C 180,E1 -4065.928,E2 -4065.928} C_VEL
LIN {X 0,Y 537.94,Z 525.991,A -85,B 0,C 180,E1 -4068.668,E2 -4068.668} C_VEL
LIN {X 0,Y 538.013,Z 516.789,A -85,B 0,C 180,E1 -4071.455,E2 -4071.455} C_VEL
LIN {X 0,Y 538.137,Z 507.622,A -85,B 0,C 180,E1 -4074.292,E2 -4074.292} C_VEL
LIN {X 0,Y 538.319,Z 498.6,A -85,B 0,C 180,E1 -4077.19,E2 -4077.19} C_VEL
LIN {X 0,Y 538.541,Z 490.023,A -85,B 0,C 180,E1 -4080.136,E2 -4080.136} C_VEL
LIN {X 0,Y 538.746,Z 482.994,A -85,B 0,C 180,E1 -4082.777,E2 -4082.777} C_VEL
LIN {X 0,Y 538.025,Z 478.282,A -85,B 0,C 180,E1 -4084.854,E2 -4084.854} C_VEL
LIN {X 0,Y 537.996,Z 478.284,A -85,B 0,C 180,E1 -4087.878,E2 -4087.878} C_VEL
LIN {X 0,Y 538.053,Z 478.276,A -85,B 0,C 180,E1 -4090.776,E2 -4090.776} C_VEL
LIN {X 0,Y 538.033,Z 478.278,A -85,B 0,C 180,E1 -4094.075,E2 -4094.075} C_VEL
LIN {X 0,Y 538.027,Z 478.278,A -85,B 0,C 180,E1 -4097.215,E2 -4097.215} C_VEL
LIN {X 0,Y 538.026,Z 478.28,A -85,B 0,C 180,E1 -4100.203,E2 -4100.203} C_VEL
LIN {X 0,Y 538.027,Z 478.282,A -85,B 0,C 180,E1 -4103.067,E2 -4103.067} C_VEL
LIN {X 0,Y 538.021,Z 478.282,A -85,B 0,C 180,E1 -4105.827,E2 -4105.827} C_VEL
LIN {X 0,Y 537.916,Z 478.297,A -85,B 0,C 180,E1 -4108.13,E2 -4108.13} C_VEL
LIN {X 0,Y 537.843,Z 480.694,A -85,B 0,C 180,E1 -4110.228,E2 -4110.228} C_VEL
LIN {X 0,Y 537.783,Z 483.932,A -85,B 0,C 180,E1 -4112.781,E2 -4112.781} C_VEL
LIN {X 0,Y 537.723,Z 487.164,A -85,B 0,C 180,E1 -4115.277,E2 -4115.277} C_VEL
LIN {X 0,Y 537.656,Z 491.437,A -85,B 0,C 180,E1 -4118.531,E2 -4118.531} C_VEL
LIN {X 0,Y 537.63,Z 494.674,A -85,B 0,C 180,E1 -4120.925,E2 -4120.925} C_VEL
LIN {X 0,Y 537.569,Z 498.86,A -85,B 0,C 180,E1 -4124.065,E2 -4124.065} C_VEL
LIN {X 0,Y 537.527,Z 502.03,A -85,B 0,C 180,E1 -4126.388,E2 -4126.388} C_VEL
LIN {X 0,Y 537.508,Z 506.711,A -85,B 0,C 180,E1 -4129.572,E2 -4129.572} C_VEL
LIN {X 0,Y 538.525,Z 516.532,A -85,B 0,C 180,E1 -4129.9,E2 -4129.9} C_VEL
LIN {X 0,Y 538.384,Z 526.504,A -85,B 0,C 180,E1 -4130.325,E2 -4130.325} C_VEL
LIN {X 0,Y 538.237,Z 535.012,A -85,B 0,C 180,E1 -4130.796,E2 -4130.796} C_VEL
LIN {X 0,Y 538.134,Z 543.181,A -85,B 0,C 180,E1 -4131.362,E2 -4131.362} C_VEL
LIN {X 0,Y 537.979,Z 550.934,A -85,B 0,C 180,E1 -4132.022,E2 -4132.022} C_VEL
LIN {X 0,Y 537.856,Z 559.035,A -85,B 0,C 180,E1 -4132.869,E2 -4132.869} C_VEL
LIN {X 0,Y 537.813,Z 565.894,A -85,B 0,C 180,E1 -4133.771,E2 -4133.771} C_VEL
LIN {X 0,Y 537.606,Z 571.757,A -85,B 0,C 180,E1 -4134.75,E2 -4134.75} C_VEL
LIN {X 0,Y 537.622,Z 576.967,A -85,B 0,C 180,E1 -4135.877,E2 -4135.877} C_VEL
LIN {X 0,Y 537.596,Z 579.649,A -85,B 0,C 180,E1 -4136.627,E2 -4136.627} C_VEL
LIN {X 0,Y 537.489,Z 582.583,A -85,B 0,C 180,E1 -4137.752,E2 -4137.752} C_VEL
LIN {X 0,Y 537.451,Z 583.872,A -85,B 0,C 180,E1 -4138.501,E2 -4138.501} C_VEL
LIN {X 0,Y 537.439,Z 584.688,A -85,B 0,C 180,E1 -4139.251,E2 -4139.251} C_VEL
LIN {X 0,Y 537.438,Z 584.996,A -85,B 0,C 180,E1 -4140,E2 -4140} C_VEL
LIN {X 0,Y 537.441,Z 584.726,A -85,B 0,C 180,E1 -4140.749,E2 -4140.749} C_VEL
LIN {X 0,Y 537.451,Z 583.988,A -85,B 0,C 180,E1 -4141.499,E2 -4141.499} C_VEL
LIN {X 0,Y 537.49,Z 582.778,A -85,B 0,C 180,E1 -4142.248,E2 -4142.248} C_VEL
LIN {X 0,Y 537.584,Z 579.925,A -85,B 0,C 180,E1 -4143.373,E2 -4143.373} C_VEL
LIN {X 0,Y 537.622,Z 577.331,A -85,B 0,C 180,E1 -4144.123,E2 -4144.123} C_VEL
LIN {X 0,Y 537.602,Z 572.217,A -85,B 0,C 180,E1 -4145.251,E2 -4145.251} C_VEL
LIN {X 0,Y 537.804,Z 566.508,A -85,B 0,C 180,E1 -4146.223,E2 -4146.223} C_VEL
LIN {X 0,Y 537.852,Z 559.817,A -85,B 0,C 180,E1 -4147.131,E2 -4147.131} C_VEL
LIN {X 0,Y 537.981,Z 550.878,A -85,B 0,C 180,E1 -4148.073,E2 -4148.073} C_VEL
LIN {X 0,Y 538.143,Z 543.116,A -85,B 0,C 180,E1 -4148.732,E2 -4148.732} C_VEL
LIN {X 0,Y 538.253,Z 534.934,A -85,B 0,C 180,E1 -4149.299,E2 -4149.299} C_VEL
LIN {X 0,Y 538.428,Z 526.403,A -85,B 0,C 180,E1 -4149.77,E2 -4149.77} C_VEL
LIN {X 0,Y 538.521,Z 515.149,A -85,B 0,C 180,E1 -4150.243,E2 -4150.243} C_VEL
LIN {X 0,Y 537.515,Z 506.515,A -85,B 0,C 180,E1 -4150.524,E2 -4150.524} C_VEL
LIN {X 0,Y 537.535,Z 502.809,A -85,B 0,C 180,E1 -4152.842,E2 -4152.842} C_VEL
LIN {X 0,Y 537.57,Z 499.223,A -85,B 0,C 180,E1 -4155.158,E2 -4155.158} C_VEL
LIN {X 0,Y 537.571,Z 494.559,A -85,B 0,C 180,E1 -4158.286,E2 -4158.286} C_VEL
LIN {X 0,Y 537.605,Z 491.093,A -85,B 0,C 180,E1 -4160.669,E2 -4160.669} C_VEL
LIN {X 0,Y 537.633,Z 487.438,A -85,B 0,C 180,E1 -4163.089,E2 -4163.089} C_VEL
LIN {X 0,Y 537.701,Z 483.681,A -85,B 0,C 180,E1 -4165.595,E2 -4165.595} C_VEL
LIN {X 0,Y 537.783,Z 481.248,A -85,B 0,C 180,E1 -4167.294,E2 -4167.294} C_VEL
LIN {X 0,Y 537.8,Z 487.346,A -85,B 0,C 180,E1 -4169.774,E2 -4169.774} C_VEL
LIN {X 0,Y 537.85,Z 493.856,A -85,B 0,C 180,E1 -4172.394,E2 -4172.394} C_VEL
LIN {X 0,Y 537.728,Z 500.197,A -85,B 0,C 180,E1 -4175.105,E2 -4175.105} C_VEL
LIN {X 0,Y 537.727,Z 503.188,A -85,B 0,C 180,E1 -4176.361,E2 -4176.361} C_VEL
LIN {X 0,Y 537.07,Z 504.697,A -85,B 0,C 180,E1 -4176.965,E2 -4176.965} C_VEL
LIN {X 0,Y 534.165,Z 507.292,A -85,B 0,C 180,E1 -4177.941,E2 -4177.941} C_VEL
LIN {X 0,Y 531.709,Z 509.381,A -85,B 0,C 180,E1 -4178.727,E2 -4178.727} C_VEL
LIN {X 0,Y 530.671,Z 510.926,A -85,B 0,C 180,E1 -4179.335,E2 -4179.335} C_VEL
LIN {X 0,Y 530.597,Z 511.429,A -85,B 0,C 180,E1 -4179.542,E2 -4179.542} C_VEL
LIN {X 0,Y 530.524,Z 518.321,A -85,B 0,C 180,E1 -4182.502,E2 -4182.502} C_VEL
LIN {X 0,Y 530.508,Z 525.033,A -85,B 0,C 180,E1 -4185.402,E2 -4185.402} C_VEL
LIN {X 0,Y 531.567,Z 534.465,A -85,B 0,C 180,E1 -4185.693,E2 -4185.693} C_VEL
LIN {X 0,Y 531.423,Z 545.9,A -85,B 0,C 180,E1 -4186.159,E2 -4186.159} C_VEL
LIN {X 0,Y 531.195,Z 556.172,A -85,B 0,C 180,E1 -4186.746,E2 -4186.746} C_VEL
LIN {X 0,Y 531.082,Z 563.844,A -85,B 0,C 180,E1 -4187.296,E2 -4187.296} C_VEL
LIN {X 0,Y 530.952,Z 570.831,A -85,B 0,C 180,E1 -4187.9,E2 -4187.9} C_VEL
LIN {X 0,Y 530.798,Z 578.193,A -85,B 0,C 180,E1 -4188.678,E2 -4188.678} C_VEL
LIN {X 0,Y 530.677,Z 584.817,A -85,B 0,C 180,E1 -4189.539,E2 -4189.539} C_VEL
LIN {X 0,Y 530.633,Z 589.082,A -85,B 0,C 180,E1 -4190.191,E2 -4190.191} C_VEL
LIN {X 0,Y 530.559,Z 593.408,A -85,B 0,C 180,E1 -4190.993,E2 -4190.993} C_VEL
LIN {X 0,Y 530.493,Z 597.629,A -85,B 0,C 180,E1 -4191.972,E2 -4191.972} C_VEL
LIN {X 0,Y 530.416,Z 601.005,A -85,B 0,C 180,E1 -4193.023,E2 -4193.023} C_VEL
LIN {X 0,Y 530.372,Z 603.064,A -85,B 0,C 180,E1 -4193.932,E2 -4193.932} C_VEL
LIN {X 0,Y 530.384,Z 604.683,A -85,B 0,C 180,E1 -4195.264,E2 -4195.264} C_VEL
LIN {X 0,Y 530.377,Z 604.968,A -85,B 0,C 180,E1 -4196.183,E2 -4196.183} C_VEL
LIN {X 0,Y 530.358,Z 604.53,A -85,B 0,C 180,E1 -4197.09,E2 -4197.09} C_VEL
LIN {X 0,Y 530.387,Z 603.334,A -85,B 0,C 180,E1 -4198,E2 -4198} C_VEL
LIN {X 0,Y 530.466,Z 601.422,A -85,B 0,C 180,E1 -4198.888,E2 -4198.888} C_VEL
LIN {X 0,Y 530.485,Z 597.262,A -85,B 0,C 180,E1 -4200.21,E2 -4200.21} C_VEL
LIN {X 0,Y 530.549,Z 592.652,A -85,B 0,C 180,E1 -4201.242,E2 -4201.242} C_VEL
LIN {X 0,Y 530.635,Z 587.379,A -85,B 0,C 180,E1 -4202.168,E2 -4202.168} C_VEL
LIN {X 0,Y 530.727,Z 581.322,A -85,B 0,C 180,E1 -4203.028,E2 -4203.028} C_VEL
LIN {X 0,Y 530.867,Z 573.863,A -85,B 0,C 180,E1 -4203.884,E2 -4203.884} C_VEL
LIN {X 0,Y 530.994,Z 567.12,A -85,B 0,C 180,E1 -4204.522,E2 -4204.522} C_VEL
LIN {X 0,Y 531.16,Z 558.908,A -85,B 0,C 180,E1 -4205.159,E2 -4205.159} C_VEL
LIN {X 0,Y 531.269,Z 550.489,A -85,B 0,C 180,E1 -4205.685,E2 -4205.685} C_VEL
LIN {X 0,Y 531.448,Z 543.084,A -85,B 0,C 180,E1 -4206.059,E2 -4206.059} C_VEL
LIN {X 0,Y 531.462,Z 532.962,A -85,B 0,C 180,E1 -4206.444,E2 -4206.444} C_VEL
LIN {X 0,Y 530.471,Z 525.293,A -85,B 0,C 180,E1 -4206.684,E2 -4206.684} C_VEL
LIN {X 0,Y 530.499,Z 518.375,A -85,B 0,C 180,E1 -4209.852,E2 -4209.852} C_VEL
LIN {X 0,Y 530.577,Z 512.674,A -85,B 0,C 180,E1 -4212.499,E2 -4212.499} C_VEL
LIN {X 0,Y 530.665,Z 506.103,A -85,B 0,C 180,E1 -4215.426,E2 -4215.426} C_VEL
LIN {X 0,Y 530.776,Z 499.224,A -85,B 0,C 180,E1 -4218.544,E2 -4218.544} C_VEL
LIN {X 0,Y 530.713,Z 492.467,A -85,B 0,C 180,E1 -4221.624,E2 -4221.624} C_VEL
LIN {X 0,Y 530.75,Z 487.31,A -85,B 0,C 180,E1 -4223.919,E2 -4223.919} C_VEL
LIN {X 0,Y 530.753,Z 482.148,A -85,B 0,C 180,E1 -4226.203,E2 -4226.203} C_VEL
LIN {X 0,Y 530.773,Z 479.186,A -85,B 0,C 180,E1 -4227.533,E2 -4227.533} C_VEL
LIN {X 0,Y 531.154,Z 479.137,A -85,B 0,C 180,E1 -4229.241,E2 -4229.241} C_VEL
LIN {X 0,Y 531.143,Z 479.137,A -85,B 0,C 180,E1 -4232.275,E2 -4232.275} C_VEL
LIN {X 0,Y 531.125,Z 479.141,A -85,B 0,C 180,E1 -4235.314,E2 -4235.314} C_VEL
LIN {X 0,Y 531.055,Z 479.149,A -85,B 0,C 180,E1 -4238.37,E2 -4238.37} C_VEL
LIN {X 0,Y 531.053,Z 479.148,A -85,B 0,C 180,E1 -4241.672,E2 -4241.672} C_VEL
LIN {X 0,Y 531.032,Z 479.151,A -85,B 0,C 180,E1 -4244.955,E2 -4244.955} C_VEL
LIN {X 0,Y 531.018,Z 479.152,A -85,B 0,C 180,E1 -4247.722,E2 -4247.722} C_VEL
LIN {X 0,Y 531.001,Z 479.154,A -85,B 0,C 180,E1 -4250.937,E2 -4250.937} C_VEL
LIN {X 0,Y 530.981,Z 479.16,A -85,B 0,C 180,E1 -4254.224,E2 -4254.224} C_VEL
LIN {X 0,Y 531.012,Z 479.154,A -85,B 0,C 180,E1 -4256.743,E2 -4256.743} C_VEL
LIN {X 0,Y 530.994,Z 479.156,A -85,B 0,C 180,E1 -4259.321,E2 -4259.321} C_VEL
LIN {X 0,Y 530.981,Z 479.158,A -85,B 0,C 180,E1 -4262.103,E2 -4262.103} C_VEL
LIN {X 0,Y 530.989,Z 479.158,A -85,B 0,C 180,E1 -4264.854,E2 -4264.854} C_VEL
LIN {X 0,Y 530.967,Z 479.16,A -85,B 0,C 180,E1 -4267.507,E2 -4267.507} C_VEL
LIN {X 0,Y 530.983,Z 479.158,A -85,B 0,C 180,E1 -4270.432,E2 -4270.432} C_VEL
LIN {X 0,Y 530.965,Z 479.16,A -85,B 0,C 180,E1 -4273.494,E2 -4273.494} C_VEL
LIN {X 0,Y 530.966,Z 479.162,A -85,B 0,C 180,E1 -4276.505,E2 -4276.505} C_VEL
LIN {X 0,Y 531.008,Z 479.154,A -85,B 0,C 180,E1 -4279.569,E2 -4279.569} C_VEL
LIN {X 0,Y 530.966,Z 479.161,A -85,B 0,C 180,E1 -4282.577,E2 -4282.577} C_VEL
LIN {X 0,Y 530.981,Z 479.157,A -85,B 0,C 180,E1 -4285.309,E2 -4285.309} C_VEL
LIN {X 0,Y 530.982,Z 479.158,A -85,B 0,C 180,E1 -4288.033,E2 -4288.033} C_VEL
LIN {X 0,Y 530.988,Z 479.158,A -85,B 0,C 180,E1 -4290.874,E2 -4290.874} C_VEL
LIN {X 0,Y 531.011,Z 479.156,A -85,B 0,C 180,E1 -4293.257,E2 -4293.257} C_VEL
LIN {X 0,Y 530.995,Z 479.156,A -85,B 0,C 180,E1 -4295.957,E2 -4295.957} C_VEL
LIN {X 0,Y 531.001,Z 479.156,A -85,B 0,C 180,E1 -4299.062,E2 -4299.062} C_VEL
LIN {X 0,Y 531.015,Z 479.154,A -85,B 0,C 180,E1 -4302.278,E2 -4302.278} C_VEL
LIN {X 0,Y 531.018,Z 479.153,A -85,B 0,C 180,E1 -4305.436,E2 -4305.436} C_VEL
LIN {X 0,Y 531.047,Z 479.151,A -85,B 0,C 180,E1 -4308.55,E2 -4308.55} C_VEL
LIN {X 0,Y 531.055,Z 479.148,A -85,B 0,C 180,E1 -4311.629,E2 -4311.629} C_VEL
LIN {X 0,Y 531.12,Z 479.14,A -85,B 0,C 180,E1 -4314.685,E2 -4314.685} C_VEL
LIN {X 0,Y 531.14,Z 479.139,A -85,B 0,C 180,E1 -4317.725,E2 -4317.725} C_VEL
LIN {X 0,Y 531.152,Z 479.135,A -85,B 0,C 180,E1 -4320.758,E2 -4320.758} C_VEL
LIN {X 0,Y 531.107,Z 479.142,A -85,B 0,C 180,E1 -4323.034,E2 -4323.034} C_VEL
LIN {X 0,Y 531.084,Z 479.147,A -85,B 0,C 180,E1 -4326.077,E2 -4326.077} C_VEL
LIN {X 0,Y 531.031,Z 479.151,A -85,B 0,C 180,E1 -4329.138,E2 -4329.138} C_VEL
LIN {X 0,Y 531.039,Z 479.151,A -85,B 0,C 180,E1 -4332.225,E2 -4332.225} C_VEL
LIN {X 0,Y 530.994,Z 479.156,A -85,B 0,C 180,E1 -4335.35,E2 -4335.35} C_VEL
LIN {X 0,Y 531.015,Z 479.154,A -85,B 0,C 180,E1 -4337.722,E2 -4337.722} C_VEL
LIN {X 0,Y 530.998,Z 479.155,A -85,B 0,C 180,E1 -4340.938,E2 -4340.938} C_VEL
LIN {X 0,Y 530.978,Z 479.158,A -85,B 0,C 180,E1 -4344.225,E2 -4344.225} C_VEL
LIN {X 0,Y 531.003,Z 479.154,A -85,B 0,C 180,E1 -4346.744,E2 -4346.744} C_VEL
LIN {X 0,Y 530.998,Z 479.155,A -85,B 0,C 180,E1 -4349.322,E2 -4349.322} C_VEL
LIN {X 0,Y 530.978,Z 479.16,A -85,B 0,C 180,E1 -4352.103,E2 -4352.103} C_VEL
LIN {X 0,Y 530.987,Z 479.158,A -85,B 0,C 180,E1 -4354.854,E2 -4354.854} C_VEL
LIN {X 0,Y 530.964,Z 479.16,A -85,B 0,C 180,E1 -4357.508,E2 -4357.508} C_VEL
LIN {X 0,Y 530.981,Z 479.159,A -85,B 0,C 180,E1 -4360.433,E2 -4360.433} C_VEL
LIN {X 0,Y 530.97,Z 479.159,A -85,B 0,C 180,E1 -4363.283,E2 -4363.283} C_VEL
LIN {X 0,Y 530.984,Z 479.157,A -85,B 0,C 180,E1 -4365.621,E2 -4365.621} C_VEL
LIN {X 0,Y 531.006,Z 479.155,A -85,B 0,C 180,E1 -4368.566,E2 -4368.566} C_VEL
LIN {X 0,Y 530.967,Z 479.161,A -85,B 0,C 180,E1 -4371.346,E2 -4371.346} C_VEL
LIN {X 0,Y 530.982,Z 479.159,A -85,B 0,C 180,E1 -4374.383,E2 -4374.383} C_VEL
LIN {X 0,Y 531.021,Z 479.304,A -85,B 0,C 180,E1 -4377.085,E2 -4377.085} C_VEL
LIN {X 0,Y 531.721,Z 483.448,A -85,B 0,C 180,E1 -4378.528,E2 -4378.528} C_VEL
LIN {X 0,Y 531.646,Z 490.215,A -85,B 0,C 180,E1 -4380.747,E2 -4380.747} C_VEL
LIN {X 0,Y 531.441,Z 498.2,A -85,B 0,C 180,E1 -4383.281,E2 -4383.281} C_VEL
LIN {X 0,Y 531.234,Z 507.847,A -85,B 0,C 180,E1 -4386.256,E2 -4386.256} C_VEL
LIN {X 0,Y 531.088,Z 517.203,A -85,B 0,C 180,E1 -4389.066,E2 -4389.066} C_VEL
LIN {X 0,Y 530.897,Z 526.738,A -85,B 0,C 180,E1 -4391.875,E2 -4391.875} C_VEL
LIN {X 0,Y 530.786,Z 536.453,A -85,B 0,C 180,E1 -4394.644,E2 -4394.644} C_VEL
LIN {X 0,Y 530.682,Z 547.513,A -85,B 0,C 180,E1 -4397.767,E2 -4397.767} C_VEL
LIN {X 0,Y 530.615,Z 552.978,A -85,B 0,C 180,E1 -4399.314,E2 -4399.314} C_VEL
LIN {X 0,Y 531.571,Z 562.917,A -85,B 0,C 180,E1 -4399.599,E2 -4399.599} C_VEL
LIN {X 0,Y 531.445,Z 573.615,A -85,B 0,C 180,E1 -4400.005,E2 -4400.005} C_VEL
LIN {X 0,Y 531.255,Z 584.227,A -85,B 0,C 180,E1 -4400.578,E2 -4400.578} C_VEL
LIN {X 0,Y 531.153,Z 592.536,A -85,B 0,C 180,E1 -4401.152,E2 -4401.152} C_VEL
LIN {X 0,Y 530.947,Z 600.396,A -85,B 0,C 180,E1 -4401.82,E2 -4401.82} C_VEL
LIN {X 0,Y 530.789,Z 607.742,A -85,B 0,C 180,E1 -4402.583,E2 -4402.583} C_VEL
LIN {X 0,Y 530.726,Z 615.247,A -85,B 0,C 180,E1 -4403.545,E2 -4403.545} C_VEL
LIN {X 0,Y 530.597,Z 621.033,A -85,B 0,C 180,E1 -4404.49,E2 -4404.49} C_VEL
LIN {X 0,Y 530.514,Z 625.634,A -85,B 0,C 180,E1 -4405.441,E2 -4405.441} C_VEL
LIN {X 0,Y 530.525,Z 628.622,A -85,B 0,C 180,E1 -4406.203,E2 -4406.203} C_VEL
